LIN {X 0,Y 572.963,Z 565.131,A -85,B 0,C 180,E1 -2344.926,E2 -2344.926} C_VEL
LIN {X 0,Y 573.073,Z 560.098,A -85,B 0,C 180,E1 -2345.984,E2 -2345.984} C_VEL
LIN {X 0,Y 573.083,Z 553.774,A -85,B 0,C 180,E1 -2347.044,E2 -2347.044} C_VEL
LIN {X 0,Y 573.175,Z 545.853,A -85,B 0,C 180,E1 -2348.106,E2 -2348.106} C_VEL
LIN {X 0,Y 573.287,Z 536.003,A -85,B 0,C 180,E1 -2349.17,E2 -2349.17} C_VEL
LIN {X 0,Y 573.412,Z 525.681,A -85,B 0,C 180,E1 -2350.059,E2 -2350.059} C_VEL
LIN {X 0,Y 573.504,Z 514.089,A -85,B 0,C 180,E1 -2350.858,E2 -2350.858} C_VEL
LIN {X 0,Y 573.658,Z 503.195,A -85,B 0,C 180,E1 -2351.449,E2 -2351.449} C_VEL
LIN {X 0,Y 573.732,Z 492.025,A -85,B 0,C 180,E1 -2351.921,E2 -2351.921} C_VEL
LIN {X 0,Y 573.827,Z 479.262,A -85,B 0,C 180,E1 -2352.309,E2 -2352.309} C_VEL
LIN {X 0,Y 573.51,Z 474.932,A -85,B 0,C 180,E1 -2352.417,E2 -2352.417} C_VEL
LIN {X 0,Y 572.962,Z 471.67,A -85,B 0,C 180,E1 -2352.508,E2 -2352.508} C_VEL
LIN {X 0,Y 572.968,Z 468.456,A -85,B 0,C 180,E1 -2354.927,E2 -2354.927} C_VEL
LIN {X 0,Y 572.954,Z 465.205,A -85,B 0,C 180,E1 -2357.402,E2 -2357.402} C_VEL
LIN {X 0,Y 572.988,Z 461.726,A -85,B 0,C 180,E1 -2360.087,E2 -2360.087} C_VEL
LIN {X 0,Y 572.974,Z 461.271,A -85,B 0,C 180,E1 -2360.442,E2 -2360.442} C_VEL
LIN {X 0,Y 572.31,Z 460.562,A -85,B 0,C 180,E1 -2361.024,E2 -2361.024} C_VEL
LIN {X 0,Y 569.449,Z 459.504,A -85,B 0,C 180,E1 -2361.969,E2 -2361.969} C_VEL
LIN {X 0,Y 567.026,Z 458.674,A -85,B 0,C 180,E1 -2362.73,E2 -2362.73} C_VEL
LIN {X 0,Y 565.982,Z 458.008,A -85,B 0,C 180,E1 -2363.318,E2 -2363.318} C_VEL
LIN {X 0,Y 565.895,Z 457.781,A -85,B 0,C 180,E1 -2363.517,E2 -2363.517} C_VEL
LIN {X 0,Y 565.976,Z 454.39,A -85,B 0,C 180,E1 -2366.554,E2 -2366.554} C_VEL
LIN {X 0,Y 565.957,Z 451.602,A -85,B 0,C 180,E1 -2368.967,E2 -2368.967} C_VEL
LIN {X 0,Y 565.973,Z 448.685,A -85,B 0,C 180,E1 -2371.436,E2 -2371.436} C_VEL
LIN {X 0,Y 566.026,Z 445.982,A -85,B 0,C 180,E1 -2373.969,E2 -2373.969} C_VEL
LIN {X 0,Y 566.197,Z 445.959,A -85,B 0,C 180,E1 -2376.571,E2 -2376.571} C_VEL
LIN {X 0,Y 566.218,Z 445.955,A -85,B 0,C 180,E1 -2379.686,E2 -2379.686} C_VEL
LIN {X 0,Y 566.219,Z 445.953,A -85,B 0,C 180,E1 -2382.087,E2 -2382.087} C_VEL
LIN {X 0,Y 566.174,Z 445.959,A -85,B 0,C 180,E1 -2385.036,E2 -2385.036} C_VEL
LIN {X 0,Y 566.194,Z 445.96,A -85,B 0,C 180,E1 -2387.911,E2 -2387.911} C_VEL
LIN {X 0,Y 566.225,Z 445.957,A -85,B 0,C 180,E1 -2390.727,E2 -2390.727} C_VEL
LIN {X 0,Y 566.191,Z 445.96,A -85,B 0,C 180,E1 -2393.788,E2 -2393.788} C_VEL
LIN {X 0,Y 566.219,Z 445.953,A -85,B 0,C 180,E1 -2396.266,E2 -2396.266} C_VEL
LIN {X 0,Y 566.193,Z 445.958,A -85,B 0,C 180,E1 -2398.924,E2 -2398.924} C_VEL
LIN {X 0,Y 566.2,Z 445.96,A -85,B 0,C 180,E1 -2401.856,E2 -2401.856} C_VEL
LIN {X 0,Y 566.22,Z 445.953,A -85,B 0,C 180,E1 -2404.251,E2 -2404.251} C_VEL
LIN {X 0,Y 566.179,Z 445.96,A -85,B 0,C 180,E1 -2406.718,E2 -2406.718} C_VEL
LIN {X 0,Y 566.214,Z 445.958,A -85,B 0,C 180,E1 -2409.663,E2 -2409.663} C_VEL
LIN {X 0,Y 566.206,Z 445.96,A -85,B 0,C 180,E1 -2412.668,E2 -2412.668} C_VEL
LIN {X 0,Y 566.241,Z 445.953,A -85,B 0,C 180,E1 -2415.627,E2 -2415.627} C_VEL
LIN {X 0,Y 566.242,Z 445.953,A -85,B 0,C 180,E1 -2418.675,E2 -2418.675} C_VEL
LIN {X 0,Y 566.211,Z 445.954,A -85,B 0,C 180,E1 -2421.434,E2 -2421.434} C_VEL
LIN {X 0,Y 566.262,Z 445.948,A -85,B 0,C 180,E1 -2424.302,E2 -2424.302} C_VEL
LIN {X 0,Y 566.288,Z 445.946,A -85,B 0,C 180,E1 -2427.866,E2 -2427.866} C_VEL
LIN {X 0,Y 566.306,Z 445.942,A -85,B 0,C 180,E1 -2430.711,E2 -2430.711} C_VEL
LIN {X 0,Y 566.273,Z 445.951,A -85,B 0,C 180,E1 -2432.845,E2 -2432.845} C_VEL
LIN {X 0,Y 566.257,Z 445.95,A -85,B 0,C 180,E1 -2435.698,E2 -2435.698} C_VEL
LIN {X 0,Y 566.234,Z 445.951,A -85,B 0,C 180,E1 -2438.565,E2 -2438.565} C_VEL
LIN {X 0,Y 566.248,Z 445.949,A -85,B 0,C 180,E1 -2441.454,E2 -2441.454} C_VEL
LIN {X 0,Y 566.241,Z 445.95,A -85,B 0,C 180,E1 -2444.506,E2 -2444.506} C_VEL
LIN {X 0,Y 566.205,Z 445.957,A -85,B 0,C 180,E1 -2447.331,E2 -2447.331} C_VEL
LIN {X 0,Y 566.213,Z 445.956,A -85,B 0,C 180,E1 -2450.337,E2 -2450.337} C_VEL
LIN {X 0,Y 566.179,Z 445.963,A -85,B 0,C 180,E1 -2453.282,E2 -2453.282} C_VEL
LIN {X 0,Y 566.218,Z 445.953,A -85,B 0,C 180,E1 -2455.749,E2 -2455.749} C_VEL
LIN {X 0,Y 566.208,Z 445.956,A -85,B 0,C 180,E1 -2458.202,E2 -2458.202} C_VEL
LIN {X 0,Y 566.198,Z 445.961,A -85,B 0,C 180,E1 -2461.076,E2 -2461.076} C_VEL
LIN {X 0,Y 566.217,Z 445.955,A -85,B 0,C 180,E1 -2463.734,E2 -2463.734} C_VEL
LIN {X 0,Y 566.211,Z 445.954,A -85,B 0,C 180,E1 -2466.569,E2 -2466.569} C_VEL
LIN {X 0,Y 566.22,Z 445.953,A -85,B 0,C 180,E1 -2469.686,E2 -2469.686} C_VEL
LIN {X 0,Y 566.205,Z 445.954,A -85,B 0,C 180,E1 -2472.917,E2 -2472.917} C_VEL
LIN {X 0,Y 566.206,Z 445.955,A -85,B 0,C 180,E1 -2476.048,E2 -2476.048} C_VEL
LIN {X 0,Y 566.185,Z 445.957,A -85,B 0,C 180,E1 -2478.861,E2 -2478.861} C_VEL
LIN {X 0,Y 566.188,Z 445.959,A -85,B 0,C 180,E1 -2481.637,E2 -2481.637} C_VEL
LIN {X 0,Y 566.208,Z 445.96,A -85,B 0,C 180,E1 -2484.311,E2 -2484.311} C_VEL
LIN {X 0,Y 566.224,Z 445.952,A -85,B 0,C 180,E1 -2486.898,E2 -2486.898} C_VEL
LIN {X 0,Y 566.187,Z 445.959,A -85,B 0,C 180,E1 -2489.407,E2 -2489.407} C_VEL
LIN {X 0,Y 566.232,Z 445.954,A -85,B 0,C 180,E1 -2491.858,E2 -2491.858} C_VEL
LIN {X 0,Y 566.215,Z 445.954,A -85,B 0,C 180,E1 -2494.251,E2 -2494.251} C_VEL
LIN {X 0,Y 566.175,Z 445.963,A -85,B 0,C 180,E1 -2496.718,E2 -2496.718} C_VEL
LIN {X 0,Y 566.216,Z 445.956,A -85,B 0,C 180,E1 -2499.663,E2 -2499.663} C_VEL
LIN {X 0,Y 566.202,Z 445.956,A -85,B 0,C 180,E1 -2502.668,E2 -2502.668} C_VEL
LIN {X 0,Y 566.237,Z 445.951,A -85,B 0,C 180,E1 -2505.627,E2 -2505.627} C_VEL
LIN {X 0,Y 566.237,Z 445.95,A -85,B 0,C 180,E1 -2508.675,E2 -2508.675} C_VEL
LIN {X 0,Y 566.235,Z 445.952,A -85,B 0,C 180,E1 -2511.434,E2 -2511.434} C_VEL
LIN {X 0,Y 566.259,Z 445.95,A -85,B 0,C 180,E1 -2514.301,E2 -2514.301} C_VEL
LIN {X 0,Y 566.278,Z 445.946,A -85,B 0,C 180,E1 -2517.866,E2 -2517.866} C_VEL
LIN {X 0,Y 566.305,Z 445.943,A -85,B 0,C 180,E1 -2520.711,E2 -2520.711} C_VEL
LIN {X 0,Y 566.275,Z 445.946,A -85,B 0,C 180,E1 -2522.845,E2 -2522.845} C_VEL
LIN {X 0,Y 566.26,Z 445.948,A -85,B 0,C 180,E1 -2525.698,E2 -2525.698} C_VEL
LIN {X 0,Y 566.229,Z 445.952,A -85,B 0,C 180,E1 -2528.566,E2 -2528.566} C_VEL
LIN {X 0,Y 566.244,Z 445.952,A -85,B 0,C 180,E1 -2531.454,E2 -2531.454} C_VEL
LIN {X 0,Y 566.236,Z 445.954,A -85,B 0,C 180,E1 -2534.507,E2 -2534.507} C_VEL
LIN {X 0,Y 566.201,Z 445.96,A -85,B 0,C 180,E1 -2537.332,E2 -2537.332} C_VEL
LIN {X 0,Y 566.216,Z 445.957,A -85,B 0,C 180,E1 -2540.337,E2 -2540.337} C_VEL
LIN {X 0,Y 566.19,Z 445.96,A -85,B 0,C 180,E1 -2543.404,E2 -2543.404} C_VEL
LIN {X 0,Y 566.215,Z 445.954,A -85,B 0,C 180,E1 -2545.749,E2 -2545.749} C_VEL
LIN {X 0,Y 566.203,Z 445.96,A -85,B 0,C 180,E1 -2548.202,E2 -2548.202} C_VEL
LIN {X 0,Y 566.192,Z 445.958,A -85,B 0,C 180,E1 -2551.077,E2 -2551.077} C_VEL
LIN {X 0,Y 566.213,Z 445.954,A -85,B 0,C 180,E1 -2553.734,E2 -2553.734} C_VEL
LIN {X 0,Y 566.216,Z 445.954,A -85,B 0,C 180,E1 -2556.569,E2 -2556.569} C_VEL
LIN {X 0,Y 566.216,Z 445.954,A -85,B 0,C 180,E1 -2559.686,E2 -2559.686} C_VEL
LIN {X 0,Y 566.216,Z 445.956,A -85,B 0,C 180,E1 -2562.087,E2 -2562.087} C_VEL
LIN {X 0,Y 566.17,Z 445.961,A -85,B 0,C 180,E1 -2565.036,E2 -2565.036} C_VEL
LIN {X 0,Y 566.191,Z 445.958,A -85,B 0,C 180,E1 -2567.911,E2 -2567.911} C_VEL
LIN {X 0,Y 566.223,Z 445.954,A -85,B 0,C 180,E1 -2570.727,E2 -2570.727} C_VEL
LIN {X 0,Y 566.236,Z 445.985,A -85,B 0,C 180,E1 -2572.989,E2 -2572.989} C_VEL
LIN {X 0,Y 566.82,Z 449.872,A -85,B 0,C 180,E1 -2574.356,E2 -2574.356} C_VEL
LIN {X 0,Y 566.804,Z 456.508,A -85,B 0,C 180,E1 -2576.554,E2 -2576.554} C_VEL
LIN {X 0,Y 566.648,Z 465.558,A -85,B 0,C 180,E1 -2579.435,E2 -2579.435} C_VEL
LIN {X 0,Y 566.506,Z 476.288,A -85,B 0,C 180,E1 -2582.676,E2 -2582.676} C_VEL
LIN {X 0,Y 566.4,Z 485.661,A -85,B 0,C 180,E1 -2585.438,E2 -2585.438} C_VEL
LIN {X 0,Y 566.323,Z 494.93,A -85,B 0,C 180,E1 -2588.143,E2 -2588.143} C_VEL
LIN {X 0,Y 566.185,Z 505.521,A -85,B 0,C 180,E1 -2591.172,E2 -2591.172} C_VEL
LIN {X 0,Y 566.116,Z 516.112,A -85,B 0,C 180,E1 -2594.15,E2 -2594.15} C_VEL
LIN {X 0,Y 566.058,Z 525.379,A -85,B 0,C 180,E1 -2596.721,E2 -2596.721} C_VEL
LIN {X 0,Y 566.033,Z 527.531,A -85,B 0,C 180,E1 -2597.314,E2 -2597.314} C_VEL
LIN {X 0,Y 566.941,Z 534.376,A -85,B 0,C 180,E1 -2597.471,E2 -2597.471} C_VEL
LIN {X 0,Y 566.856,Z 546.503,A -85,B 0,C 180,E1 -2597.787,E2 -2597.787} C_VEL
LIN {X 0,Y 566.719,Z 558.32,A -85,B 0,C 180,E1 -2598.229,E2 -2598.229} C_VEL
LIN {X 0,Y 566.571,Z 570.729,A -85,B 0,C 180,E1 -2598.854,E2 -2598.854} C_VEL
LIN {X 0,Y 566.418,Z 581.483,A -85,B 0,C 180,E1 -2599.545,E2 -2599.545} C_VEL
LIN {X 0,Y 566.301,Z 591.648,A -85,B 0,C 180,E1 -2600.355,E2 -2600.355} C_VEL
LIN {X 0,Y 566.166,Z 600.788,A -85,B 0,C 180,E1 -2601.254,E2 -2601.254} C_VEL
LIN {X 0,Y 566.08,Z 609.691,A -85,B 0,C 180,E1 -2602.33,E2 -2602.33} C_VEL
LIN {X 0,Y 565.967,Z 616.956,A -85,B 0,C 180,E1 -2603.422,E2 -2603.422} C_VEL
LIN {X 0,Y 566.004,Z 621.681,A -85,B 0,C 180,E1 -2604.299,E2 -2604.299} C_VEL
LIN {X 0,Y 565.933,Z 626.373,A -85,B 0,C 180,E1 -2605.37,E2 -2605.37} C_VEL
LIN {X 0,Y 565.927,Z 629.958,A -85,B 0,C 180,E1 -2606.44,E2 -2606.44} C_VEL
LIN {X 0,Y 565.878,Z 631.809,A -85,B 0,C 180,E1 -2607.153,E2 -2607.153} C_VEL
LIN {X 0,Y 565.846,Z 634.186,A -85,B 0,C 180,E1 -2608.577,E2 -2608.577} C_VEL
LIN {X 0,Y 565.839,Z 635,A -85,B 0,C 180,E1 -2610,E2 -2610} C_VEL
LIN {X 0,Y 565.846,Z 634.186,A -85,B 0,C 180,E1 -2611.424,E2 -2611.424} C_VEL
LIN {X 0,Y 565.878,Z 631.809,A -85,B 0,C 180,E1 -2612.848,E2 -2612.848} C_VEL
LIN {X 0,Y 565.926,Z 628.895,A -85,B 0,C 180,E1 -2613.917,E2 -2613.917} C_VEL
LIN {X 0,Y 565.878,Z 624.948,A -85,B 0,C 180,E1 -2614.988,E2 -2614.988} C_VEL
LIN {X 0,Y 566.002,Z 619.866,A -85,B 0,C 180,E1 -2616.059,E2 -2616.059} C_VEL
LIN {X 0,Y 566.04,Z 613.467,A -85,B 0,C 180,E1 -2617.132,E2 -2617.132} C_VEL
LIN {X 0,Y 566.134,Z 605.477,A -85,B 0,C 180,E1 -2618.208,E2 -2618.208} C_VEL
LIN {X 0,Y 566.229,Z 597.334,A -85,B 0,C 180,E1 -2619.106,E2 -2619.106} C_VEL
LIN {X 0,Y 566.343,Z 587.399,A -85,B 0,C 180,E1 -2620.005,E2 -2620.005} C_VEL
LIN {X 0,Y 566.535,Z 576.295,A -85,B 0,C 180,E1 -2620.807,E2 -2620.807} C_VEL
LIN {X 0,Y 566.613,Z 565.174,A -85,B 0,C 180,E1 -2621.447,E2 -2621.447} C_VEL
LIN {X 0,Y 566.75,Z 552.98,A -85,B 0,C 180,E1 -2621.988,E2 -2621.988} C_VEL
LIN {X 0,Y 566.881,Z 540.169,A -85,B 0,C 180,E1 -2622.394,E2 -2622.394} C_VEL
LIN {X 0,Y 566.748,Z 532.075,A -85,B 0,C 180,E1 -2622.579,E2 -2622.579} C_VEL
LIN {X 0,Y 566.033,Z 527.529,A -85,B 0,C 180,E1 -2622.686,E2 -2622.686} C_VEL
LIN {X 0,Y 566.091,Z 517.435,A -85,B 0,C 180,E1 -2625.481,E2 -2625.481} C_VEL
LIN {X 0,Y 566.167,Z 506.844,A -85,B 0,C 180,E1 -2628.454,E2 -2628.454} C_VEL
LIN {X 0,Y 566.245,Z 497.576,A -85,B 0,C 180,E1 -2631.096,E2 -2631.096} C_VEL
LIN {X 0,Y 566.362,Z 488.309,A -85,B 0,C 180,E1 -2633.784,E2 -2633.784} C_VEL
LIN {X 0,Y 566.426,Z 480.094,A -85,B 0,C 180,E1 -2636.134,E2 -2636.134} C_VEL
LIN {X 0,Y 566.448,Z 471.713,A -85,B 0,C 180,E1 -2638.557,E2 -2638.557} C_VEL
LIN {X 0,Y 566.56,Z 463.235,A -85,B 0,C 180,E1 -2641.138,E2 -2641.138} C_VEL
LIN {X 0,Y 566.718,Z 455.161,A -85,B 0,C 180,E1 -2643.81,E2 -2643.81} C_VEL
LIN {X 0,Y 566.858,Z 450.195,A -85,B 0,C 180,E1 -2645.642,E2 -2645.642} C_VEL
LIN {X 0,Y 566.22,Z 445.959,A -85,B 0,C 180,E1 -2647.571,E2 -2647.571} C_VEL
LIN {X 0,Y 566.231,Z 445.957,A -85,B 0,C 180,E1 -2650.197,E2 -2650.197} C_VEL
LIN {X 0,Y 566.204,Z 445.958,A -85,B 0,C 180,E1 -2653.054,E2 -2653.054} C_VEL
LIN {X 0,Y 566.206,Z 445.96,A -85,B 0,C 180,E1 -2656.048,E2 -2656.048} C_VEL
LIN {X 0,Y 566.215,Z 445.958,A -85,B 0,C 180,E1 -2658.864,E2 -2658.864} C_VEL
LIN {X 0,Y 566.194,Z 445.959,A -85,B 0,C 180,E1 -2661.637,E2 -2661.637} C_VEL
LIN {X 0,Y 566.137,Z 445.967,A -85,B 0,C 180,E1 -2664.306,E2 -2664.306} C_VEL
LIN {X 0,Y 566.127,Z 446.063,A -85,B 0,C 180,E1 -2665.176,E2 -2665.176} C_VEL
LIN {X 0,Y 566.103,Z 448.7,A -85,B 0,C 180,E1 -2667.735,E2 -2667.735} C_VEL
LIN {X 0,Y 566.046,Z 451.422,A -85,B 0,C 180,E1 -2670.357,E2 -2670.357} C_VEL
LIN {X 0,Y 566.001,Z 454.553,A -85,B 0,C 180,E1 -2673.448,E2 -2673.448} C_VEL
LIN {X 0,Y 565.923,Z 456.995,A -85,B 0,C 180,E1 -2675.807,E2 -2675.807} C_VEL
LIN {X 0,Y 565.906,Z 460.651,A -85,B 0,C 180,E1 -2678.891,E2 -2678.891} C_VEL
LIN {X 0,Y 565.866,Z 464.495,A -85,B 0,C 180,E1 -2681.911,E2 -2681.911} C_VEL
LIN {X 0,Y 565.89,Z 468.338,A -85,B 0,C 180,E1 -2684.882,E2 -2684.882} C_VEL
LIN {X 0,Y 565.873,Z 471.671,A -85,B 0,C 180,E1 -2687.424,E2 -2687.424} C_VEL
LIN {X 0,Y 566.904,Z 479.284,A -85,B 0,C 180,E1 -2687.629,E2 -2687.629} C_VEL
LIN {X 0,Y 566.781,Z 491.783,A -85,B 0,C 180,E1 -2688.013,E2 -2688.013} C_VEL
LIN {X 0,Y 566.661,Z 504.301,A -85,B 0,C 180,E1 -2688.554,E2 -2688.554} C_VEL
LIN {X 0,Y 566.543,Z 515.586,A -85,B 0,C 180,E1 -2689.193,E2 -2689.193} C_VEL
LIN {X 0,Y 566.341,Z 526.843,A -85,B 0,C 180,E1 -2689.995,E2 -2689.995} C_VEL
LIN {X 0,Y 566.238,Z 536.892,A -85,B 0,C 180,E1 -2690.895,E2 -2690.895} C_VEL
LIN {X 0,Y 566.113,Z 546.592,A -85,B 0,C 180,E1 -2691.972,E2 -2691.972} C_VEL
LIN {X 0,Y 566.05,Z 553.16,A -85,B 0,C 180,E1 -2692.868,E2 -2692.868} C_VEL
LIN {X 0,Y 566.003,Z 559.628,A -85,B 0,C 180,E1 -2693.942,E2 -2693.942} C_VEL
LIN {X 0,Y 565.878,Z 564.765,A -85,B 0,C 180,E1 -2695.013,E2 -2695.013} C_VEL
LIN {X 0,Y 565.926,Z 568.754,A -85,B 0,C 180,E1 -2696.084,E2 -2696.084} C_VEL
LIN {X 0,Y 565.878,Z 571.702,A -85,B 0,C 180,E1 -2697.153,E2 -2697.153} C_VEL
LIN {X 0,Y 565.839,Z 573.129,A -85,B 0,C 180,E1 -2697.865,E2 -2697.865} C_VEL
LIN {X 0,Y 565.841,Z 574.756,A -85,B 0,C 180,E1 -2699.289,E2 -2699.289} C_VEL
LIN {X 0,Y 565.839,Z 574.996,A -85,B 0,C 180,E1 -2700,E2 -2700} C_VEL
LIN {X 0,Y 565.841,Z 574.814,A -85,B 0,C 180,E1 -2700.712,E2 -2700.712} C_VEL
LIN {X 0,Y 565.838,Z 573.269,A -85,B 0,C 180,E1 -2702.136,E2 -2702.136} C_VEL
LIN {X 0,Y 565.878,Z 571.907,A -85,B 0,C 180,E1 -2702.848,E2 -2702.848} C_VEL
LIN {X 0,Y 565.926,Z 569.029,A -85,B 0,C 180,E1 -2703.917,E2 -2703.917} C_VEL
LIN {X 0,Y 565.878,Z 565.128,A -85,B 0,C 180,E1 -2704.988,E2 -2704.988} C_VEL
LIN {X 0,Y 565.988,Z 560.095,A -85,B 0,C 180,E1 -2706.059,E2 -2706.059} C_VEL
LIN {X 0,Y 566.031,Z 553.771,A -85,B 0,C 180,E1 -2707.133,E2 -2707.133} C_VEL
LIN {X 0,Y 566.128,Z 545.848,A -85,B 0,C 180,E1 -2708.208,E2 -2708.208} C_VEL
LIN {X 0,Y 566.249,Z 535.997,A -85,B 0,C 180,E1 -2709.285,E2 -2709.285} C_VEL
LIN {X 0,Y 566.413,Z 525.675,A -85,B 0,C 180,E1 -2710.184,E2 -2710.184} C_VEL
LIN {X 0,Y 566.519,Z 514.394,A -85,B 0,C 180,E1 -2710.973,E2 -2710.973} C_VEL
LIN {X 0,Y 566.688,Z 503.183,A -85,B 0,C 180,E1 -2711.592,E2 -2711.592} C_VEL
LIN {X 0,Y 566.786,Z 492.009,A -85,B 0,C 180,E1 -2712.069,E2 -2712.069} C_VEL
LIN {X 0,Y 566.896,Z 479.239,A -85,B 0,C 180,E1 -2712.462,E2 -2712.462} C_VEL
LIN {X 0,Y 565.878,Z 471.669,A -85,B 0,C 180,E1 -2712.667,E2 -2712.667} C_VEL
LIN {X 0,Y 565.891,Z 468.455,A -85,B 0,C 180,E1 -2715.118,E2 -2715.118} C_VEL
LIN {X 0,Y 565.868,Z 464.61,A -85,B 0,C 180,E1 -2718.089,E2 -2718.089} C_VEL
LIN {X 0,Y 565.906,Z 460.764,A -85,B 0,C 180,E1 -2721.11,E2 -2721.11} C_VEL
LIN {X 0,Y 565.895,Z 457.781,A -85,B 0,C 180,E1 -2723.517,E2 -2723.517} C_VEL
LIN {X 0,Y 565.218,Z 457.167,A -85,B 0,C 180,E1 -2724.107,E2 -2724.107} C_VEL
LIN {X 0,Y 562.35,Z 456.326,A -85,B 0,C 180,E1 -2725.068,E2 -2725.068} C_VEL
LIN {X 0,Y 559.956,Z 455.672,A -85,B 0,C 180,E1 -2725.842,E2 -2725.842} C_VEL
LIN {X 0,Y 558.962,Z 455.108,A -85,B 0,C 180,E1 -2726.438,E2 -2726.438} C_VEL
LIN {X 0,Y 558.898,Z 454.896,A -85,B 0,C 180,E1 -2726.639,E2 -2726.639} C_VEL
LIN {X 0,Y 558.904,Z 451.659,A -85,B 0,C 180,E1 -2729.368,E2 -2729.368} C_VEL
LIN {X 0,Y 558.901,Z 448.772,A -85,B 0,C 180,E1 -2731.88,E2 -2731.88} C_VEL
LIN {X 0,Y 558.928,Z 446.866,A -85,B 0,C 180,E1 -2733.591,E2 -2733.591} C_VEL
LIN {X 0,Y 559.141,Z 446.837,A -85,B 0,C 180,E1 -2736.444,E2 -2736.444} C_VEL
LIN {X 0,Y 559.177,Z 446.83,A -85,B 0,C 180,E1 -2738.934,E2 -2738.934} C_VEL
LIN {X 0,Y 559.182,Z 446.83,A -85,B 0,C 180,E1 -2742.137,E2 -2742.137} C_VEL
LIN {X 0,Y 559.14,Z 446.834,A -85,B 0,C 180,E1 -2745.261,E2 -2745.261} C_VEL
LIN {X 0,Y 559.168,Z 446.832,A -85,B 0,C 180,E1 -2748.23,E2 -2748.23} C_VEL
LIN {X 0,Y 559.182,Z 446.831,A -85,B 0,C 180,E1 -2751.192,E2 -2751.192} C_VEL
LIN {X 0,Y 559.146,Z 446.837,A -85,B 0,C 180,E1 -2753.789,E2 -2753.789} C_VEL
LIN {X 0,Y 559.169,Z 446.831,A -85,B 0,C 180,E1 -2756.425,E2 -2756.425} C_VEL
LIN {X 0,Y 559.157,Z 446.834,A -85,B 0,C 180,E1 -2758.981,E2 -2758.981} C_VEL
LIN {X 0,Y 559.151,Z 446.837,A -85,B 0,C 180,E1 -2761.623,E2 -2761.623} C_VEL
LIN {X 0,Y 559.187,Z 446.829,A -85,B 0,C 180,E1 -2763.903,E2 -2763.903} C_VEL
LIN {X 0,Y 559.149,Z 446.837,A -85,B 0,C 180,E1 -2766.571,E2 -2766.571} C_VEL
LIN {X 0,Y 559.183,Z 446.833,A -85,B 0,C 180,E1 -2769.395,E2 -2769.395} C_VEL
LIN {X 0,Y 559.148,Z 446.834,A -85,B 0,C 180,E1 -2771.686,E2 -2771.686} C_VEL
LIN {X 0,Y 559.167,Z 446.834,A -85,B 0,C 180,E1 -2773.948,E2 -2773.948} C_VEL
LIN {X 0,Y 559.178,Z 446.831,A -85,B 0,C 180,E1 -2776.184,E2 -2776.184} C_VEL
LIN {X 0,Y 559.201,Z 446.83,A -85,B 0,C 180,E1 -2779.133,E2 -2779.133} C_VEL
LIN {X 0,Y 559.198,Z 446.833,A -85,B 0,C 180,E1 -2782.053,E2 -2782.053} C_VEL
LIN {X 0,Y 559.256,Z 446.824,A -85,B 0,C 180,E1 -2784.953,E2 -2784.953} C_VEL
LIN {X 0,Y 559.259,Z 446.821,A -85,B 0,C 180,E1 -2787.839,E2 -2787.839} C_VEL
LIN {X 0,Y 559.277,Z 446.818,A -85,B 0,C 180,E1 -2790.72,E2 -2790.72} C_VEL
LIN {X 0,Y 559.24,Z 446.827,A -85,B 0,C 180,E1 -2792.881,E2 -2792.881} C_VEL
LIN {X 0,Y 559.225,Z 446.826,A -85,B 0,C 180,E1 -2795.77,E2 -2795.77} C_VEL
LIN {X 0,Y 559.193,Z 446.829,A -85,B 0,C 180,E1 -2798.674,E2 -2798.674} C_VEL
LIN {X 0,Y 559.212,Z 446.826,A -85,B 0,C 180,E1 -2801.6,E2 -2801.6} C_VEL
LIN {X 0,Y 559.207,Z 446.826,A -85,B 0,C 180,E1 -2804.595,E2 -2804.595} C_VEL
LIN {X 0,Y 559.164,Z 446.832,A -85,B 0,C 180,E1 -2807.557,E2 -2807.557} C_VEL
LIN {X 0,Y 559.171,Z 446.834,A -85,B 0,C 180,E1 -2809.837,E2 -2809.837} C_VEL
LIN {X 0,Y 559.146,Z 446.835,A -85,B 0,C 180,E1 -2812.153,E2 -2812.153} C_VEL
LIN {X 0,Y 559.181,Z 446.83,A -85,B 0,C 180,E1 -2815.298,E2 -2815.298} C_VEL
LIN {X 0,Y 559.173,Z 446.831,A -85,B 0,C 180,E1 -2818.381,E2 -2818.381} C_VEL
LIN {X 0,Y 559.153,Z 446.836,A -85,B 0,C 180,E1 -2821.273,E2 -2821.273} C_VEL
LIN {X 0,Y 559.172,Z 446.835,A -85,B 0,C 180,E1 -2823.949,E2 -2823.949} C_VEL
LIN {X 0,Y 559.147,Z 446.838,A -85,B 0,C 180,E1 -2827.108,E2 -2827.108} C_VEL
LIN {X 0,Y 559.165,Z 446.833,A -85,B 0,C 180,E1 -2829.941,E2 -2829.941} C_VEL
LIN {X 0,Y 559.16,Z 446.831,A -85,B 0,C 180,E1 -2832.743,E2 -2832.743} C_VEL
LIN {X 0,Y 559.159,Z 446.833,A -85,B 0,C 180,E1 -2835.76,E2 -2835.76} C_VEL
LIN {X 0,Y 559.192,Z 446.833,A -85,B 0,C 180,E1 -2838.232,E2 -2838.232} C_VEL
LIN {X 0,Y 559.177,Z 446.834,A -85,B 0,C 180,E1 -2841.191,E2 -2841.191} C_VEL
LIN {X 0,Y 559.173,Z 446.831,A -85,B 0,C 180,E1 -2843.791,E2 -2843.791} C_VEL
LIN {X 0,Y 559.165,Z 446.832,A -85,B 0,C 180,E1 -2846.425,E2 -2846.425} C_VEL
LIN {X 0,Y 559.162,Z 446.836,A -85,B 0,C 180,E1 -2848.981,E2 -2848.981} C_VEL
LIN {X 0,Y 559.171,Z 446.831,A -85,B 0,C 180,E1 -2851.618,E2 -2851.618} C_VEL
LIN {X 0,Y 559.183,Z 446.833,A -85,B 0,C 180,E1 -2853.903,E2 -2853.903} C_VEL
LIN {X 0,Y 559.145,Z 446.837,A -85,B 0,C 180,E1 -2856.571,E2 -2856.571} C_VEL
LIN {X 0,Y 559.182,Z 446.83,A -85,B 0,C 180,E1 -2859.395,E2 -2859.395} C_VEL
LIN {X 0,Y 559.146,Z 446.838,A -85,B 0,C 180,E1 -2861.685,E2 -2861.685} C_VEL
LIN {X 0,Y 559.169,Z 446.831,A -85,B 0,C 180,E1 -2863.948,E2 -2863.948} C_VEL
LIN {X 0,Y 559.175,Z 446.836,A -85,B 0,C 180,E1 -2866.184,E2 -2866.184} C_VEL
LIN {X 0,Y 559.196,Z 446.83,A -85,B 0,C 180,E1 -2869.133,E2 -2869.133} C_VEL
LIN {X 0,Y 559.207,Z 446.828,A -85,B 0,C 180,E1 -2872.053,E2 -2872.053} C_VEL
LIN {X 0,Y 559.256,Z 446.82,A -85,B 0,C 180,E1 -2874.953,E2 -2874.953} C_VEL
LIN {X 0,Y 559.25,Z 446.821,A -85,B 0,C 180,E1 -2877.839,E2 -2877.839} C_VEL
LIN {X 0,Y 559.275,Z 446.819,A -85,B 0,C 180,E1 -2880.72,E2 -2880.72} C_VEL
LIN {X 0,Y 559.241,Z 446.822,A -85,B 0,C 180,E1 -2882.881,E2 -2882.881} C_VEL
LIN {X 0,Y 559.229,Z 446.824,A -85,B 0,C 180,E1 -2885.77,E2 -2885.77} C_VEL
LIN {X 0,Y 559.188,Z 446.829,A -85,B 0,C 180,E1 -2888.674,E2 -2888.674} C_VEL
LIN {X 0,Y 559.207,Z 446.828,A -85,B 0,C 180,E1 -2891.6,E2 -2891.6} C_VEL
LIN {X 0,Y 559.201,Z 446.829,A -85,B 0,C 180,E1 -2894.595,E2 -2894.595} C_VEL
LIN {X 0,Y 559.161,Z 446.836,A -85,B 0,C 180,E1 -2897.557,E2 -2897.557} C_VEL
LIN {X 0,Y 559.174,Z 446.831,A -85,B 0,C 180,E1 -2899.837,E2 -2899.837} C_VEL
LIN {X 0,Y 559.144,Z 446.839,A -85,B 0,C 180,E1 -2902.153,E2 -2902.153} C_VEL
LIN {X 0,Y 559.177,Z 446.835,A -85,B 0,C 180,E1 -2905.298,E2 -2905.298} C_VEL
LIN {X 0,Y 559.182,Z 446.83,A -85,B 0,C 180,E1 -2907.712,E2 -2907.712} C_VEL
LIN {X 0,Y 559.155,Z 446.835,A -85,B 0,C 180,E1 -2910.183,E2 -2910.183} C_VEL
LIN {X 0,Y 559.158,Z 446.834,A -85,B 0,C 180,E1 -2912.715,E2 -2912.715} C_VEL
LIN {X 0,Y 559.15,Z 446.834,A -85,B 0,C 180,E1 -2915.323,E2 -2915.323} C_VEL
LIN {X 0,Y 559.134,Z 446.837,A -85,B 0,C 180,E1 -2918.018,E2 -2918.018} C_VEL
LIN {X 0,Y 559.163,Z 446.837,A -85,B 0,C 180,E1 -2920.812,E2 -2920.812} C_VEL
LIN {X 0,Y 559.164,Z 446.836,A -85,B 0,C 180,E1 -2923.732,E2 -2923.732} C_VEL
LIN {X 0,Y 559.146,Z 446.839,A -85,B 0,C 180,E1 -2926.804,E2 -2926.804} C_VEL
LIN {X 0,Y 559.175,Z 446.832,A -85,B 0,C 180,E1 -2929.189,E2 -2929.189} C_VEL
LIN {X 0,Y 559.136,Z 446.84,A -85,B 0,C 180,E1 -2931.983,E2 -2931.983} C_VEL
LIN {X 0,Y 559.215,Z 447.004,A -85,B 0,C 180,E1 -2932.8,E2 -2932.8} C_VEL
LIN {X 0,Y 559.892,Z 452.465,A -85,B 0,C 180,E1 -2934.731,E2 -2934.731} C_VEL
LIN {X 0,Y 559.772,Z 460.095,A -85,B 0,C 180,E1 -2937.267,E2 -2937.267} C_VEL
LIN {X 0,Y 559.625,Z 468.857,A -85,B 0,C 180,E1 -2940.058,E2 -2940.058} C_VEL
LIN {X 0,Y 559.467,Z 478.897,A -85,B 0,C 180,E1 -2943.113,E2 -2943.113} C_VEL
LIN {X 0,Y 559.379,Z 488.262,A -85,B 0,C 180,E1 -2945.9,E2 -2945.9} C_VEL
LIN {X 0,Y 559.233,Z 497.577,A -85,B 0,C 180,E1 -2948.626,E2 -2948.626} C_VEL
LIN {X 0,Y 559.134,Z 506.845,A -85,B 0,C 180,E1 -2951.306,E2 -2951.306} C_VEL
LIN {X 0,Y 559.055,Z 517.436,A -85,B 0,C 180,E1 -2954.319,E2 -2954.319} C_VEL
LIN {X 0,Y 558.955,Z 527.531,A -85,B 0,C 180,E1 -2957.151,E2 -2957.151} C_VEL
LIN {X 0,Y 560.015,Z 535.515,A -85,B 0,C 180,E1 -2957.336,E2 -2957.336} C_VEL
LIN {X 0,Y 559.897,Z 547.879,A -85,B 0,C 180,E1 -2957.679,E2 -2957.679} C_VEL
LIN {X 0,Y 559.759,Z 560.285,A -85,B 0,C 180,E1 -2958.172,E2 -2958.172} C_VEL
LIN {X 0,Y 559.608,Z 572.583,A -85,B 0,C 180,E1 -2958.822,E2 -2958.822} C_VEL
LIN {X 0,Y 559.425,Z 583.926,A -85,B 0,C 180,E1 -2959.596,E2 -2959.596} C_VEL
LIN {X 0,Y 559.243,Z 593.602,A -85,B 0,C 180,E1 -2960.415,E2 -2960.415} C_VEL
LIN {X 0,Y 559.127,Z 602.414,A -85,B 0,C 180,E1 -2961.325,E2 -2961.325} C_VEL
LIN {X 0,Y 558.996,Z 611.003,A -85,B 0,C 180,E1 -2962.414,E2 -2962.414} C_VEL
LIN {X 0,Y 558.884,Z 618.688,A -85,B 0,C 180,E1 -2963.649,E2 -2963.649} C_VEL
LIN {X 0,Y 558.869,Z 623.366,A -85,B 0,C 180,E1 -2964.588,E2 -2964.588} C_VEL
LIN {X 0,Y 558.868,Z 627.678,A -85,B 0,C 180,E1 -2965.673,E2 -2965.673} C_VEL
LIN {X 0,Y 558.836,Z 629.958,A -85,B 0,C 180,E1 -2966.395,E2 -2966.395} C_VEL
LIN {X 0,Y 558.799,Z 631.808,A -85,B 0,C 180,E1 -2967.117,E2 -2967.117} C_VEL
LIN {X 0,Y 558.745,Z 634.185,A -85,B 0,C 180,E1 -2968.559,E2 -2968.559} C_VEL
LIN {X 0,Y 558.74,Z 635,A -85,B 0,C 180,E1 -2970,E2 -2970} C_VEL
LIN {X 0,Y 558.745,Z 634.186,A -85,B 0,C 180,E1 -2971.442,E2 -2971.442} C_VEL
LIN {X 0,Y 558.799,Z 631.81,A -85,B 0,C 180,E1 -2972.884,E2 -2972.884} C_VEL
LIN {X 0,Y 558.843,Z 628.895,A -85,B 0,C 180,E1 -2973.966,E2 -2973.966} C_VEL
LIN {X 0,Y 558.799,Z 624.948,A -85,B 0,C 180,E1 -2975.051,E2 -2975.051} C_VEL
LIN {X 0,Y 558.921,Z 619.866,A -85,B 0,C 180,E1 -2976.136,E2 -2976.136} C_VEL
LIN {X 0,Y 558.977,Z 613.467,A -85,B 0,C 180,E1 -2977.223,E2 -2977.223} C_VEL
LIN {X 0,Y 559.099,Z 605.477,A -85,B 0,C 180,E1 -2978.312,E2 -2978.312} C_VEL
LIN {X 0,Y 559.195,Z 597.333,A -85,B 0,C 180,E1 -2979.221,E2 -2979.221} C_VEL
LIN {X 0,Y 559.351,Z 587.398,A -85,B 0,C 180,E1 -2980.131,E2 -2980.131} C_VEL
LIN {X 0,Y 559.538,Z 576.398,A -85,B 0,C 180,E1 -2980.937,E2 -2980.937} C_VEL
LIN {X 0,Y 559.672,Z 564.458,A -85,B 0,C 180,E1 -2981.628,E2 -2981.628} C_VEL
LIN {X 0,Y 559.824,Z 551.762,A -85,B 0,C 180,E1 -2982.185,E2 -2982.185} C_VEL
LIN {X 0,Y 559.974,Z 538.339,A -85,B 0,C 180,E1 -2982.596,E2 -2982.596} C_VEL
LIN {X 0,Y 559.749,Z 532.507,A -85,B 0,C 180,E1 -2982.73,E2 -2982.73} C_VEL
LIN {X 0,Y 558.955,Z 527.529,A -85,B 0,C 180,E1 -2982.85,E2 -2982.85} C_VEL
LIN {X 0,Y 559.055,Z 517.435,A -85,B 0,C 180,E1 -2985.681,E2 -2985.681} C_VEL
LIN {X 0,Y 559.134,Z 506.844,A -85,B 0,C 180,E1 -2988.695,E2 -2988.695} C_VEL
LIN {X 0,Y 559.227,Z 496.916,A -85,B 0,C 180,E1 -2991.567,E2 -2991.567} C_VEL
LIN {X 0,Y 559.345,Z 488.126,A -85,B 0,C 180,E1 -2994.102,E2 -2994.102} C_VEL
LIN {X 0,Y 559.42,Z 478.359,A -85,B 0,C 180,E1 -2996.89,E2 -2996.89} C_VEL
LIN {X 0,Y 559.529,Z 468.262,A -85,B 0,C 180,E1 -2999.925,E2 -2999.925} C_VEL
LIN {X 0,Y 559.677,Z 459.655,A -85,B 0,C 180,E1 -3002.718,E2 -3002.718} C_VEL
LIN {X 0,Y 559.896,Z 452.496,A -85,B 0,C 180,E1 -3005.323,E2 -3005.323} C_VEL
LIN {X 0,Y 559.691,Z 449.63,A -85,B 0,C 180,E1 -3006.52,E2 -3006.52} C_VEL
LIN {X 0,Y 559.169,Z 446.837,A -85,B 0,C 180,E1 -3007.907,E2 -3007.907} C_VEL
LIN {X 0,Y 559.177,Z 446.834,A -85,B 0,C 180,E1 -3010.811,E2 -3010.811} C_VEL
LIN {X 0,Y 559.144,Z 446.84,A -85,B 0,C 180,E1 -3013.734,E2 -3013.734} C_VEL
LIN {X 0,Y 559.172,Z 446.834,A -85,B 0,C 180,E1 -3016.801,E2 -3016.801} C_VEL
LIN {X 0,Y 559.18,Z 446.833,A -85,B 0,C 180,E1 -3019.19,E2 -3019.19} C_VEL
LIN {X 0,Y 559.139,Z 446.839,A -85,B 0,C 180,E1 -3021.983,E2 -3021.983} C_VEL
LIN {X 0,Y 559.075,Z 446.849,A -85,B 0,C 180,E1 -3024.672,E2 -3024.672} C_VEL
LIN {X 0,Y 559.059,Z 448.217,A -85,B 0,C 180,E1 -3026.418,E2 -3026.418} C_VEL
LIN {X 0,Y 559.03,Z 450.796,A -85,B 0,C 180,E1 -3028.973,E2 -3028.973} C_VEL
LIN {X 0,Y 558.95,Z 453.54,A -85,B 0,C 180,E1 -3031.661,E2 -3031.661} C_VEL
LIN {X 0,Y 558.896,Z 456.578,A -85,B 0,C 180,E1 -3034.688,E2 -3034.688} C_VEL
LIN {X 0,Y 558.816,Z 459.044,A -85,B 0,C 180,E1 -3037.053,E2 -3037.053} C_VEL
LIN {X 0,Y 558.789,Z 461.613,A -85,B 0,C 180,E1 -3039.38,E2 -3039.38} C_VEL
LIN {X 0,Y 558.764,Z 464.495,A -85,B 0,C 180,E1 -3041.673,E2 -3041.673} C_VEL
LIN {X 0,Y 558.773,Z 467.378,A -85,B 0,C 180,E1 -3043.936,E2 -3043.936} C_VEL
LIN {X 0,Y 558.782,Z 470.261,A -85,B 0,C 180,E1 -3046.174,E2 -3046.174} C_VEL
LIN {X 0,Y 558.784,Z 471.672,A -85,B 0,C 180,E1 -3047.262,E2 -3047.262} C_VEL
LIN {X 0,Y 559.972,Z 480.22,A -85,B 0,C 180,E1 -3047.497,E2 -3047.497} C_VEL
LIN {X 0,Y 559.835,Z 492.301,A -85,B 0,C 180,E1 -3047.88,E2 -3047.88} C_VEL
LIN {X 0,Y 559.688,Z 504.311,A -85,B 0,C 180,E1 -3048.41,E2 -3048.41} C_VEL
LIN {X 0,Y 559.566,Z 515.668,A -85,B 0,C 180,E1 -3049.061,E2 -3049.061} C_VEL
LIN {X 0,Y 559.356,Z 526.851,A -85,B 0,C 180,E1 -3049.869,E2 -3049.869} C_VEL
LIN {X 0,Y 559.21,Z 536.897,A -85,B 0,C 180,E1 -3050.779,E2 -3050.779} C_VEL
LIN {X 0,Y 559.05,Z 546.596,A -85,B 0,C 180,E1 -3051.87,E2 -3051.87} C_VEL
LIN {X 0,Y 558.971,Z 554.456,A -85,B 0,C 180,E1 -3052.977,E2 -3052.977} C_VEL
LIN {X 0,Y 558.936,Z 561.455,A -85,B 0,C 180,E1 -3054.227,E2 -3054.227} C_VEL
LIN {X 0,Y 558.826,Z 566.195,A -85,B 0,C 180,E1 -3055.311,E2 -3055.311} C_VEL
LIN {X 0,Y 558.837,Z 569.828,A -85,B 0,C 180,E1 -3056.395,E2 -3056.395} C_VEL
LIN {X 0,Y 558.799,Z 571.704,A -85,B 0,C 180,E1 -3057.117,E2 -3057.117} C_VEL
LIN {X 0,Y 558.745,Z 573.129,A -85,B 0,C 180,E1 -3057.838,E2 -3057.838} C_VEL
LIN {X 0,Y 558.742,Z 574.757,A -85,B 0,C 180,E1 -3059.279,E2 -3059.279} C_VEL
LIN {X 0,Y 558.74,Z 574.996,A -85,B 0,C 180,E1 -3060,E2 -3060} C_VEL
LIN {X 0,Y 558.741,Z 574.814,A -85,B 0,C 180,E1 -3060.721,E2 -3060.721} C_VEL
LIN {X 0,Y 558.745,Z 573.267,A -85,B 0,C 180,E1 -3062.163,E2 -3062.163} C_VEL
LIN {X 0,Y 558.8,Z 571.905,A -85,B 0,C 180,E1 -3062.884,E2 -3062.884} C_VEL
LIN {X 0,Y 558.844,Z 569.028,A -85,B 0,C 180,E1 -3063.966,E2 -3063.966} C_VEL
LIN {X 0,Y 558.798,Z 565.126,A -85,B 0,C 180,E1 -3065.051,E2 -3065.051} C_VEL
LIN {X 0,Y 558.908,Z 560.093,A -85,B 0,C 180,E1 -3066.136,E2 -3066.136} C_VEL
LIN {X 0,Y 558.973,Z 553.767,A -85,B 0,C 180,E1 -3067.223,E2 -3067.223} C_VEL
LIN {X 0,Y 559.091,Z 545.843,A -85,B 0,C 180,E1 -3068.312,E2 -3068.312} C_VEL
LIN {X 0,Y 559.224,Z 535.99,A -85,B 0,C 180,E1 -3069.403,E2 -3069.403} C_VEL
LIN {X 0,Y 559.399,Z 525.669,A -85,B 0,C 180,E1 -3070.313,E2 -3070.313} C_VEL
LIN {X 0,Y 559.533,Z 514.701,A -85,B 0,C 180,E1 -3071.091,E2 -3071.091} C_VEL
LIN {X 0,Y 559.709,Z 504.45,A -85,B 0,C 180,E1 -3071.673,E2 -3071.673} C_VEL
LIN {X 0,Y 559.818,Z 492.957,A -85,B 0,C 180,E1 -3072.185,E2 -3072.185} C_VEL
LIN {X 0,Y 559.963,Z 480.13,A -85,B 0,C 180,E1 -3072.596,E2 -3072.596} C_VEL
LIN {X 0,Y 558.769,Z 471.668,A -85,B 0,C 180,E1 -3072.831,E2 -3072.831} C_VEL
LIN {X 0,Y 558.808,Z 468.454,A -85,B 0,C 180,E1 -3075.314,E2 -3075.314} C_VEL
LIN {X 0,Y 558.774,Z 465.57,A -85,B 0,C 180,E1 -3077.57,E2 -3077.57} C_VEL
LIN {X 0,Y 558.794,Z 462.686,A -85,B 0,C 180,E1 -3079.852,E2 -3079.852} C_VEL
LIN {X 0,Y 558.797,Z 459.864,A -85,B 0,C 180,E1 -3082.168,E2 -3082.168} C_VEL
LIN {X 0,Y 558.849,Z 456.561,A -85,B 0,C 180,E1 -3085.114,E2 -3085.114} C_VEL
LIN {X 0,Y 558.898,Z 454.896,A -85,B 0,C 180,E1 -3086.639,E2 -3086.639} C_VEL
LIN {X 0,Y 558.29,Z 454.271,A -85,B 0,C 180,E1 -3087.237,E2 -3087.237} C_VEL
LIN {X 0,Y 555.484,Z 453.323,A -85,B 0,C 180,E1 -3088.209,E2 -3088.209} C_VEL
LIN {X 0,Y 553.053,Z 452.561,A -85,B 0,C 180,E1 -3088.992,E2 -3088.992} C_VEL
LIN {X 0,Y 551.967,Z 451.934,A -85,B 0,C 180,E1 -3089.595,E2 -3089.595} C_VEL
LIN {X 0,Y 551.858,Z 451.708,A -85,B 0,C 180,E1 -3089.799,E2 -3089.799} C_VEL
LIN {X 0,Y 551.845,Z 448.341,A -85,B 0,C 180,E1 -3092.802,E2 -3092.802} C_VEL
LIN {X 0,Y 551.837,Z 447.89,A -85,B 0,C 180,E1 -3093.205,E2 -3093.205} C_VEL
LIN {X 0,Y 552.03,Z 447.724,A -85,B 0,C 180,E1 -3095.432,E2 -3095.432} C_VEL
LIN {X 0,Y 552.1,Z 447.712,A -85,B 0,C 180,E1 -3097.886,E2 -3097.886} C_VEL
LIN {X 0,Y 552.115,Z 447.71,A -85,B 0,C 180,E1 -3100.481,E2 -3100.481} C_VEL
LIN {X 0,Y 552.125,Z 447.71,A -85,B 0,C 180,E1 -3103.485,E2 -3103.485} C_VEL
LIN {X 0,Y 552.112,Z 447.711,A -85,B 0,C 180,E1 -3106.576,E2 -3106.576} C_VEL
LIN {X 0,Y 552.115,Z 447.713,A -85,B 0,C 180,E1 -3109.519,E2 -3109.519} C_VEL
LIN {X 0,Y 552.098,Z 447.717,A -85,B 0,C 180,E1 -3112.336,E2 -3112.336} C_VEL
LIN {X 0,Y 552.093,Z 447.713,A -85,B 0,C 180,E1 -3115.051,E2 -3115.051} C_VEL
LIN {X 0,Y 552.121,Z 447.71,A -85,B 0,C 180,E1 -3117.681,E2 -3117.681} C_VEL
LIN {X 0,Y 552.113,Z 447.715,A -85,B 0,C 180,E1 -3120.235,E2 -3120.235} C_VEL
LIN {X 0,Y 552.143,Z 447.709,A -85,B 0,C 180,E1 -3123,E2 -3123} C_VEL
LIN {X 0,Y 552.12,Z 447.712,A -85,B 0,C 180,E1 -3125.161,E2 -3125.161} C_VEL
LIN {X 0,Y 552.132,Z 447.709,A -85,B 0,C 180,E1 -3128.337,E2 -3128.337} C_VEL
LIN {X 0,Y 552.157,Z 447.706,A -85,B 0,C 180,E1 -3130.674,E2 -3130.674} C_VEL
LIN {X 0,Y 552.118,Z 447.71,A -85,B 0,C 180,E1 -3133.737,E2 -3133.737} C_VEL
LIN {X 0,Y 552.142,Z 447.71,A -85,B 0,C 180,E1 -3136.004,E2 -3136.004} C_VEL
LIN {X 0,Y 552.169,Z 447.707,A -85,B 0,C 180,E1 -3138.993,E2 -3138.993} C_VEL
LIN {X 0,Y 552.153,Z 447.71,A -85,B 0,C 180,E1 -3141.951,E2 -3141.951} C_VEL
LIN {X 0,Y 552.231,Z 447.698,A -85,B 0,C 180,E1 -3144.889,E2 -3144.889} C_VEL
LIN {X 0,Y 552.23,Z 447.697,A -85,B 0,C 180,E1 -3147.812,E2 -3147.812} C_VEL
LIN {X 0,Y 552.247,Z 447.693,A -85,B 0,C 180,E1 -3150.729,E2 -3150.729} C_VEL
LIN {X 0,Y 552.207,Z 447.703,A -85,B 0,C 180,E1 -3152.918,E2 -3152.918} C_VEL
LIN {X 0,Y 552.195,Z 447.703,A -85,B 0,C 180,E1 -3155.844,E2 -3155.844} C_VEL
LIN {X 0,Y 552.164,Z 447.705,A -85,B 0,C 180,E1 -3158.785,E2 -3158.785} C_VEL
LIN {X 0,Y 552.169,Z 447.704,A -85,B 0,C 180,E1 -3161.75,E2 -3161.75} C_VEL
LIN {X 0,Y 552.142,Z 447.706,A -85,B 0,C 180,E1 -3164.748,E2 -3164.748} C_VEL
LIN {X 0,Y 552.115,Z 447.71,A -85,B 0,C 180,E1 -3167.788,E2 -3167.788} C_VEL
LIN {X 0,Y 552.132,Z 447.713,A -85,B 0,C 180,E1 -3170.101,E2 -3170.101} C_VEL
LIN {X 0,Y 552.098,Z 447.712,A -85,B 0,C 180,E1 -3172.451,E2 -3172.451} C_VEL
LIN {X 0,Y 552.161,Z 447.705,A -85,B 0,C 180,E1 -3175.35,E2 -3175.35} C_VEL
LIN {X 0,Y 552.108,Z 447.714,A -85,B 0,C 180,E1 -3178.098,E2 -3178.098} C_VEL
LIN {X 0,Y 552.109,Z 447.712,A -85,B 0,C 180,E1 -3180.609,E2 -3180.609} C_VEL
LIN {X 0,Y 552.12,Z 447.709,A -85,B 0,C 180,E1 -3183.185,E2 -3183.185} C_VEL
LIN {X 0,Y 552.104,Z 447.715,A -85,B 0,C 180,E1 -3185.842,E2 -3185.842} C_VEL
LIN {X 0,Y 552.126,Z 447.712,A -85,B 0,C 180,E1 -3189.061,E2 -3189.061} C_VEL
LIN {X 0,Y 552.124,Z 447.709,A -85,B 0,C 180,E1 -3191.446,E2 -3191.446} C_VEL
LIN {X 0,Y 552.099,Z 447.713,A -85,B 0,C 180,E1 -3194.531,E2 -3194.531} C_VEL
LIN {X 0,Y 552.135,Z 447.708,A -85,B 0,C 180,E1 -3197.584,E2 -3197.584} C_VEL
LIN {X 0,Y 552.132,Z 447.707,A -85,B 0,C 180,E1 -3200.472,E2 -3200.472} C_VEL
LIN {X 0,Y 552.118,Z 447.711,A -85,B 0,C 180,E1 -3203.315,E2 -3203.315} C_VEL
LIN {X 0,Y 552.131,Z 447.713,A -85,B 0,C 180,E1 -3205.939,E2 -3205.939} C_VEL
LIN {X 0,Y 552.122,Z 447.709,A -85,B 0,C 180,E1 -3208.54,E2 -3208.54} C_VEL
LIN {X 0,Y 552.127,Z 447.709,A -85,B 0,C 180,E1 -3211.438,E2 -3211.438} C_VEL
LIN {X 0,Y 552.132,Z 447.707,A -85,B 0,C 180,E1 -3214.355,E2 -3214.355} C_VEL
LIN {X 0,Y 552.101,Z 447.716,A -85,B 0,C 180,E1 -3216.758,E2 -3216.758} C_VEL
LIN {X 0,Y 552.123,Z 447.709,A -85,B 0,C 180,E1 -3219.12,E2 -3219.12} C_VEL
LIN {X 0,Y 552.125,Z 447.713,A -85,B 0,C 180,E1 -3221.444,E2 -3221.444} C_VEL
LIN {X 0,Y 552.119,Z 447.71,A -85,B 0,C 180,E1 -3223.737,E2 -3223.737} C_VEL
LIN {X 0,Y 552.138,Z 447.71,A -85,B 0,C 180,E1 -3226.004,E2 -3226.004} C_VEL
LIN {X 0,Y 552.164,Z 447.705,A -85,B 0,C 180,E1 -3228.993,E2 -3228.993} C_VEL
LIN {X 0,Y 552.161,Z 447.705,A -85,B 0,C 180,E1 -3231.951,E2 -3231.951} C_VEL
LIN {X 0,Y 552.23,Z 447.695,A -85,B 0,C 180,E1 -3234.889,E2 -3234.889} C_VEL
LIN {X 0,Y 552.222,Z 447.697,A -85,B 0,C 180,E1 -3237.812,E2 -3237.812} C_VEL
LIN {X 0,Y 552.245,Z 447.695,A -85,B 0,C 180,E1 -3240.729,E2 -3240.729} C_VEL
LIN {X 0,Y 552.208,Z 447.699,A -85,B 0,C 180,E1 -3242.918,E2 -3242.918} C_VEL
LIN {X 0,Y 552.2,Z 447.7,A -85,B 0,C 180,E1 -3245.844,E2 -3245.844} C_VEL
LIN {X 0,Y 552.159,Z 447.704,A -85,B 0,C 180,E1 -3248.786,E2 -3248.786} C_VEL
LIN {X 0,Y 552.164,Z 447.704,A -85,B 0,C 180,E1 -3251.75,E2 -3251.75} C_VEL
LIN {X 0,Y 552.138,Z 447.708,A -85,B 0,C 180,E1 -3254.748,E2 -3254.748} C_VEL
LIN {X 0,Y 552.112,Z 447.711,A -85,B 0,C 180,E1 -3257.788,E2 -3257.788} C_VEL
LIN {X 0,Y 552.133,Z 447.709,A -85,B 0,C 180,E1 -3260.101,E2 -3260.101} C_VEL
LIN {X 0,Y 552.095,Z 447.714,A -85,B 0,C 180,E1 -3262.451,E2 -3262.451} C_VEL
LIN {X 0,Y 552.157,Z 447.709,A -85,B 0,C 180,E1 -3265.35,E2 -3265.35} C_VEL
LIN {X 0,Y 552.121,Z 447.713,A -85,B 0,C 180,E1 -3268.098,E2 -3268.098} C_VEL
LIN {X 0,Y 552.104,Z 447.711,A -85,B 0,C 180,E1 -3270.609,E2 -3270.609} C_VEL
LIN {X 0,Y 552.116,Z 447.713,A -85,B 0,C 180,E1 -3273.186,E2 -3273.186} C_VEL
LIN {X 0,Y 552.11,Z 447.713,A -85,B 0,C 180,E1 -3275.842,E2 -3275.842} C_VEL
LIN {X 0,Y 552.122,Z 447.712,A -85,B 0,C 180,E1 -3279.061,E2 -3279.061} C_VEL
LIN {X 0,Y 552.14,Z 447.707,A -85,B 0,C 180,E1 -3281.444,E2 -3281.444} C_VEL
LIN {X 0,Y 552.096,Z 447.714,A -85,B 0,C 180,E1 -3284.532,E2 -3284.532} C_VEL
LIN {X 0,Y 552.13,Z 447.71,A -85,B 0,C 180,E1 -3287.585,E2 -3287.585} C_VEL
LIN {X 0,Y 552.136,Z 447.711,A -85,B 0,C 180,E1 -3290.473,E2 -3290.473} C_VEL
LIN {X 0,Y 552.132,Z 447.769,A -85,B 0,C 180,E1 -3292.512,E2 -3292.512} C_VEL
LIN {X 0,Y 552.927,Z 453.079,A -85,B 0,C 180,E1 -3294.437,E2 -3294.437} C_VEL
LIN {X 0,Y 552.829,Z 460.243,A -85,B 0,C 180,E1 -3296.863,E2 -3296.863} C_VEL
LIN {X 0,Y 552.648,Z 469.448,A -85,B 0,C 180,E1 -3299.855,E2 -3299.855} C_VEL
LIN {X 0,Y 552.473,Z 479.39,A -85,B 0,C 180,E1 -3302.933,E2 -3302.933} C_VEL
LIN {X 0,Y 552.325,Z 489.433,A -85,B 0,C 180,E1 -3305.972,E2 -3305.972} C_VEL
LIN {X 0,Y 552.199,Z 498.889,A -85,B 0,C 180,E1 -3308.732,E2 -3308.732} C_VEL
LIN {X 0,Y 552.085,Z 508.169,A -85,B 0,C 180,E1 -3311.443,E2 -3311.443} C_VEL
LIN {X 0,Y 551.981,Z 518.76,A -85,B 0,C 180,E1 -3314.492,E2 -3314.492} C_VEL
LIN {X 0,Y 551.909,Z 527.531,A -85,B 0,C 180,E1 -3316.984,E2 -3316.984} C_VEL
LIN {X 0,Y 553.097,Z 535.515,A -85,B 0,C 180,E1 -3317.175,E2 -3317.175} C_VEL
LIN {X 0,Y 552.972,Z 547.878,A -85,B 0,C 180,E1 -3317.522,E2 -3317.522} C_VEL
LIN {X 0,Y 552.813,Z 559.509,A -85,B 0,C 180,E1 -3317.985,E2 -3317.985} C_VEL
LIN {X 0,Y 552.633,Z 571.899,A -85,B 0,C 180,E1 -3318.638,E2 -3318.638} C_VEL
LIN {X 0,Y 552.415,Z 582.747,A -85,B 0,C 180,E1 -3319.37,E2 -3319.37} C_VEL
LIN {X 0,Y 552.232,Z 593.601,A -85,B 0,C 180,E1 -3320.292,E2 -3320.292} C_VEL
LIN {X 0,Y 552.079,Z 602.414,A -85,B 0,C 180,E1 -3321.213,E2 -3321.213} C_VEL
LIN {X 0,Y 551.949,Z 611.003,A -85,B 0,C 180,E1 -3322.317,E2 -3322.317} C_VEL
LIN {X 0,Y 551.823,Z 617.869,A -85,B 0,C 180,E1 -3323.418,E2 -3323.418} C_VEL
LIN {X 0,Y 551.804,Z 623.367,A -85,B 0,C 180,E1 -3324.519,E2 -3324.519} C_VEL
LIN {X 0,Y 551.764,Z 627.678,A -85,B 0,C 180,E1 -3325.617,E2 -3325.617} C_VEL
LIN {X 0,Y 551.75,Z 629.958,A -85,B 0,C 180,E1 -3326.349,E2 -3326.349} C_VEL
LIN {X 0,Y 551.723,Z 631.808,A -85,B 0,C 180,E1 -3327.079,E2 -3327.079} C_VEL
LIN {X 0,Y 551.645,Z 634.185,A -85,B 0,C 180,E1 -3328.54,E2 -3328.54} C_VEL
LIN {X 0,Y 551.64,Z 635,A -85,B 0,C 180,E1 -3330,E2 -3330} C_VEL
LIN {X 0,Y 551.645,Z 634.185,A -85,B 0,C 180,E1 -3331.46,E2 -3331.46} C_VEL
LIN {X 0,Y 551.723,Z 631.81,A -85,B 0,C 180,E1 -3332.921,E2 -3332.921} C_VEL
LIN {X 0,Y 551.764,Z 628.895,A -85,B 0,C 180,E1 -3334.017,E2 -3334.017} C_VEL
LIN {X 0,Y 551.724,Z 624.948,A -85,B 0,C 180,E1 -3335.116,E2 -3335.116} C_VEL
LIN {X 0,Y 551.803,Z 619.188,A -85,B 0,C 180,E1 -3336.342,E2 -3336.342} C_VEL
LIN {X 0,Y 551.926,Z 612.235,A -85,B 0,C 180,E1 -3337.5,E2 -3337.5} C_VEL
LIN {X 0,Y 552.082,Z 603.99,A -85,B 0,C 180,E1 -3338.603,E2 -3338.603} C_VEL
LIN {X 0,Y 552.201,Z 595.537,A -85,B 0,C 180,E1 -3339.524,E2 -3339.524} C_VEL
LIN {X 0,Y 552.419,Z 585.093,A -85,B 0,C 180,E1 -3340.445,E2 -3340.445} C_VEL
LIN {X 0,Y 552.59,Z 574.294,A -85,B 0,C 180,E1 -3341.213,E2 -3341.213} C_VEL
LIN {X 0,Y 552.754,Z 563.404,A -85,B 0,C 180,E1 -3341.831,E2 -3341.831} C_VEL
LIN {X 0,Y 552.902,Z 551.758,A -85,B 0,C 180,E1 -3342.34,E2 -3342.34} C_VEL
LIN {X 0,Y 553.063,Z 539.253,A -85,B 0,C 180,E1 -3342.732,E2 -3342.732} C_VEL
LIN {X 0,Y 552.905,Z 533.785,A -85,B 0,C 180,E1 -3342.864,E2 -3342.864} C_VEL
LIN {X 0,Y 551.909,Z 527.529,A -85,B 0,C 180,E1 -3343.017,E2 -3343.017} C_VEL
LIN {X 0,Y 551.996,Z 517.435,A -85,B 0,C 180,E1 -3345.887,E2 -3345.887} C_VEL
LIN {X 0,Y 552.085,Z 506.844,A -85,B 0,C 180,E1 -3348.942,E2 -3348.942} C_VEL
LIN {X 0,Y 552.185,Z 497.337,A -85,B 0,C 180,E1 -3351.702,E2 -3351.702} C_VEL
LIN {X 0,Y 552.304,Z 487.75,A -85,B 0,C 180,E1 -3354.429,E2 -3354.429} C_VEL
LIN {X 0,Y 552.409,Z 478.027,A -85,B 0,C 180,E1 -3357.259,E2 -3357.259} C_VEL
LIN {X 0,Y 552.583,Z 467.311,A -85,B 0,C 180,E1 -3360.58,E2 -3360.58} C_VEL
LIN {X 0,Y 552.751,Z 458.538,A -85,B 0,C 180,E1 -3363.579,E2 -3363.579} C_VEL
LIN {X 0,Y 552.972,Z 452.85,A -85,B 0,C 180,E1 -3365.778,E2 -3365.778} C_VEL
LIN {X 0,Y 552.234,Z 448.353,A -85,B 0,C 180,E1 -3367.904,E2 -3367.904} C_VEL
LIN {X 0,Y 552.126,Z 447.714,A -85,B 0,C 180,E1 -3368.398,E2 -3368.398} C_VEL
LIN {X 0,Y 552.132,Z 447.713,A -85,B 0,C 180,E1 -3371.445,E2 -3371.445} C_VEL
LIN {X 0,Y 552.099,Z 447.716,A -85,B 0,C 180,E1 -3374.532,E2 -3374.532} C_VEL
LIN {X 0,Y 552.135,Z 447.713,A -85,B 0,C 180,E1 -3377.585,E2 -3377.585} C_VEL
LIN {X 0,Y 552.136,Z 447.711,A -85,B 0,C 180,E1 -3380.473,E2 -3380.473} C_VEL
LIN {X 0,Y 552.105,Z 447.717,A -85,B 0,C 180,E1 -3383.318,E2 -3383.318} C_VEL
LIN {X 0,Y 552.026,Z 447.787,A -85,B 0,C 180,E1 -3385.047,E2 -3385.047} C_VEL
LIN {X 0,Y 552.005,Z 450.34,A -85,B 0,C 180,E1 -3387.674,E2 -3387.674} C_VEL
LIN {X 0,Y 551.962,Z 452.88,A -85,B 0,C 180,E1 -3390.226,E2 -3390.226} C_VEL
LIN {X 0,Y 551.86,Z 455.737,A -85,B 0,C 180,E1 -3393.058,E2 -3393.058} C_VEL
LIN {X 0,Y 551.801,Z 458.653,A -85,B 0,C 180,E1 -3395.948,E2 -3395.948} C_VEL
LIN {X 0,Y 551.723,Z 461.953,A -85,B 0,C 180,E1 -3399.104,E2 -3399.104} C_VEL
LIN {X 0,Y 551.67,Z 464.496,A -85,B 0,C 180,E1 -3401.429,E2 -3401.429} C_VEL
LIN {X 0,Y 551.708,Z 467.379,A -85,B 0,C 180,E1 -3403.725,E2 -3403.725} C_VEL
LIN {X 0,Y 551.7,Z 470.261,A -85,B 0,C 180,E1 -3405.993,E2 -3405.993} C_VEL
LIN {X 0,Y 551.674,Z 471.673,A -85,B 0,C 180,E1 -3407.095,E2 -3407.095} C_VEL
LIN {X 0,Y 553.037,Z 480.243,A -85,B 0,C 180,E1 -3407.337,E2 -3407.337} C_VEL
LIN {X 0,Y 552.878,Z 493.017,A -85,B 0,C 180,E1 -3407.753,E2 -3407.753} C_VEL
LIN {X 0,Y 552.718,Z 504.321,A -85,B 0,C 180,E1 -3408.262,E2 -3408.262} C_VEL
LIN {X 0,Y 552.582,Z 515.76,A -85,B 0,C 180,E1 -3408.927,E2 -3408.927} C_VEL
LIN {X 0,Y 552.369,Z 526.859,A -85,B 0,C 180,E1 -3409.739,E2 -3409.739} C_VEL
LIN {X 0,Y 552.174,Z 536.902,A -85,B 0,C 180,E1 -3410.661,E2 -3410.661} C_VEL
LIN {X 0,Y 552.007,Z 546.601,A -85,B 0,C 180,E1 -3411.765,E2 -3411.765} C_VEL
LIN {X 0,Y 551.895,Z 554.46,A -85,B 0,C 180,E1 -3412.886,E2 -3412.886} C_VEL
LIN {X 0,Y 551.868,Z 561.458,A -85,B 0,C 180,E1 -3414.153,E2 -3414.153} C_VEL
LIN {X 0,Y 551.725,Z 566.198,A -85,B 0,C 180,E1 -3415.251,E2 -3415.251} C_VEL
LIN {X 0,Y 551.751,Z 569.83,A -85,B 0,C 180,E1 -3416.349,E2 -3416.349} C_VEL
LIN {X 0,Y 551.724,Z 571.706,A -85,B 0,C 180,E1 -3417.079,E2 -3417.079} C_VEL
LIN {X 0,Y 551.656,Z 573.129,A -85,B 0,C 180,E1 -3417.81,E2 -3417.81} C_VEL
LIN {X 0,Y 551.642,Z 574.757,A -85,B 0,C 180,E1 -3419.27,E2 -3419.27} C_VEL
LIN {X 0,Y 551.641,Z 574.996,A -85,B 0,C 180,E1 -3420,E2 -3420} C_VEL
LIN {X 0,Y 551.642,Z 574.814,A -85,B 0,C 180,E1 -3420.73,E2 -3420.73} C_VEL
LIN {X 0,Y 551.655,Z 573.265,A -85,B 0,C 180,E1 -3422.191,E2 -3422.191} C_VEL
LIN {X 0,Y 551.724,Z 571.904,A -85,B 0,C 180,E1 -3422.921,E2 -3422.921} C_VEL
LIN {X 0,Y 551.764,Z 569.026,A -85,B 0,C 180,E1 -3424.017,E2 -3424.017} C_VEL
LIN {X 0,Y 551.723,Z 565.124,A -85,B 0,C 180,E1 -3425.116,E2 -3425.116} C_VEL
LIN {X 0,Y 551.81,Z 559.397,A -85,B 0,C 180,E1 -3426.349,E2 -3426.349} C_VEL
LIN {X 0,Y 551.926,Z 552.536,A -85,B 0,C 180,E1 -3427.5,E2 -3427.5} C_VEL
LIN {X 0,Y 552.063,Z 544.352,A -85,B 0,C 180,E1 -3428.603,E2 -3428.603} C_VEL
LIN {X 0,Y 552.197,Z 535.984,A -85,B 0,C 180,E1 -3429.524,E2 -3429.524} C_VEL
LIN {X 0,Y 552.402,Z 525.662,A -85,B 0,C 180,E1 -3430.446,E2 -3430.446} C_VEL
LIN {X 0,Y 552.583,Z 513.878,A -85,B 0,C 180,E1 -3431.286,E2 -3431.286} C_VEL
LIN {X 0,Y 552.76,Z 502.438,A -85,B 0,C 180,E1 -3431.924,E2 -3431.924} C_VEL
LIN {X 0,Y 552.93,Z 490.424,A -85,B 0,C 180,E1 -3432.432,E2 -3432.432} C_VEL
LIN {X 0,Y 552.843,Z 478.733,A -85,B 0,C 180,E1 -3432.796,E2 -3432.796} C_VEL
LIN {X 0,Y 551.673,Z 471.668,A -85,B 0,C 180,E1 -3432.999,E2 -3432.999} C_VEL
LIN {X 0,Y 551.722,Z 468.453,A -85,B 0,C 180,E1 -3435.516,E2 -3435.516} C_VEL
LIN {X 0,Y 551.685,Z 465.569,A -85,B 0,C 180,E1 -3437.803,E2 -3437.803} C_VEL
LIN {X 0,Y 551.692,Z 462.734,A -85,B 0,C 180,E1 -3440.118,E2 -3440.118} C_VEL
LIN {X 0,Y 551.728,Z 460.064,A -85,B 0,C 180,E1 -3442.467,E2 -3442.467} C_VEL
LIN {X 0,Y 551.781,Z 456.972,A -85,B 0,C 180,E1 -3445.267,E2 -3445.267} C_VEL
LIN {X 0,Y 551.808,Z 454.638,A -85,B 0,C 180,E1 -3447.291,E2 -3447.291} C_VEL
LIN {X 0,Y 551.858,Z 451.708,A -85,B 0,C 180,E1 -3449.799,E2 -3449.799} C_VEL
LIN {X 0,Y 551.136,Z 451.083,A -85,B 0,C 180,E1 -3450.405,E2 -3450.405} C_VEL
LIN {X 0,Y 548.268,Z 450.226,A -85,B 0,C 180,E1 -3451.39,E2 -3451.39} C_VEL
LIN {X 0,Y 545.88,Z 449.553,A -85,B 0,C 180,E1 -3452.184,E2 -3452.184} C_VEL
LIN {X 0,Y 544.858,Z 448.966,A -85,B 0,C 180,E1 -3452.795,E2 -3452.795} C_VEL
LIN {X 0,Y 544.774,Z 448.743,A -85,B 0,C 180,E1 -3453.002,E2 -3453.002} C_VEL
LIN {X 0,Y 544.996,Z 448.6,A -85,B 0,C 180,E1 -3455.472,E2 -3455.472} C_VEL
LIN {X 0,Y 545.054,Z 448.592,A -85,B 0,C 180,E1 -3458.136,E2 -3458.136} C_VEL
LIN {X 0,Y 545.087,Z 448.586,A -85,B 0,C 180,E1 -3460.473,E2 -3460.473} C_VEL
LIN {X 0,Y 545.084,Z 448.59,A -85,B 0,C 180,E1 -3463.107,E2 -3463.107} C_VEL
LIN {X 0,Y 545.054,Z 448.594,A -85,B 0,C 180,E1 -3466.226,E2 -3466.226} C_VEL
LIN {X 0,Y 545.087,Z 448.587,A -85,B 0,C 180,E1 -3468.886,E2 -3468.886} C_VEL
LIN {X 0,Y 545.088,Z 448.59,A -85,B 0,C 180,E1 -3470.819,E2 -3470.819} C_VEL
LIN {X 0,Y 545.048,Z 448.591,A -85,B 0,C 180,E1 -3473.62,E2 -3473.62} C_VEL
LIN {X 0,Y 545.073,Z 448.587,A -85,B 0,C 180,E1 -3476.328,E2 -3476.328} C_VEL
LIN {X 0,Y 545.07,Z 448.589,A -85,B 0,C 180,E1 -3478.952,E2 -3478.952} C_VEL
LIN {X 0,Y 545.089,Z 448.587,A -85,B 0,C 180,E1 -3481.507,E2 -3481.507} C_VEL
LIN {X 0,Y 545.102,Z 448.585,A -85,B 0,C 180,E1 -3484.491,E2 -3484.491} C_VEL
LIN {X 0,Y 545.044,Z 448.59,A -85,B 0,C 180,E1 -3487.242,E2 -3487.242} C_VEL
LIN {X 0,Y 545.123,Z 448.581,A -85,B 0,C 180,E1 -3490.415,E2 -3490.415} C_VEL
LIN {X 0,Y 545.069,Z 448.587,A -85,B 0,C 180,E1 -3493.521,E2 -3493.521} C_VEL
LIN {X 0,Y 545.102,Z 448.589,A -85,B 0,C 180,E1 -3495.82,E2 -3495.82} C_VEL
LIN {X 0,Y 545.125,Z 448.585,A -85,B 0,C 180,E1 -3498.849,E2 -3498.849} C_VEL
LIN {X 0,Y 545.102,Z 448.587,A -85,B 0,C 180,E1 -3501.846,E2 -3501.846} C_VEL
LIN {X 0,Y 545.175,Z 448.575,A -85,B 0,C 180,E1 -3504.08,E2 -3504.08} C_VEL
LIN {X 0,Y 545.174,Z 448.576,A -85,B 0,C 180,E1 -3507.044,E2 -3507.044} C_VEL
LIN {X 0,Y 545.209,Z 448.574,A -85,B 0,C 180,E1 -3510,E2 -3510} C_VEL
LIN {X 0,Y 545.174,Z 448.579,A -85,B 0,C 180,E1 -3512.956,E2 -3512.956} C_VEL
LIN {X 0,Y 545.165,Z 448.579,A -85,B 0,C 180,E1 -3515.919,E2 -3515.919} C_VEL
LIN {X 0,Y 545.123,Z 448.583,A -85,B 0,C 180,E1 -3518.9,E2 -3518.9} C_VEL
LIN {X 0,Y 545.141,Z 448.58,A -85,B 0,C 180,E1 -3521.904,E2 -3521.904} C_VEL
LIN {X 0,Y 545.091,Z 448.585,A -85,B 0,C 180,E1 -3524.943,E2 -3524.943} C_VEL
LIN {X 0,Y 545.083,Z 448.587,A -85,B 0,C 180,E1 -3528.026,E2 -3528.026} C_VEL
LIN {X 0,Y 545.098,Z 448.586,A -85,B 0,C 180,E1 -3530.372,E2 -3530.372} C_VEL
LIN {X 0,Y 545.087,Z 448.588,A -85,B 0,C 180,E1 -3533.559,E2 -3533.559} C_VEL
LIN {X 0,Y 545.083,Z 448.588,A -85,B 0,C 180,E1 -3536,E2 -3536} C_VEL
LIN {X 0,Y 545.094,Z 448.584,A -85,B 0,C 180,E1 -3538.748,E2 -3538.748} C_VEL
LIN {X 0,Y 545.062,Z 448.589,A -85,B 0,C 180,E1 -3541.678,E2 -3541.678} C_VEL
LIN {X 0,Y 545.082,Z 448.586,A -85,B 0,C 180,E1 -3544.563,E2 -3544.563} C_VEL
LIN {X 0,Y 545.042,Z 448.596,A -85,B 0,C 180,E1 -3547.303,E2 -3547.303} C_VEL
LIN {X 0,Y 545.069,Z 448.591,A -85,B 0,C 180,E1 -3550.142,E2 -3550.142} C_VEL
LIN {X 0,Y 545.082,Z 448.587,A -85,B 0,C 180,E1 -3553.106,E2 -3553.106} C_VEL
LIN {X 0,Y 545.069,Z 448.59,A -85,B 0,C 180,E1 -3556.224,E2 -3556.224} C_VEL
LIN {X 0,Y 545.091,Z 448.584,A -85,B 0,C 180,E1 -3558.886,E2 -3558.886} C_VEL
LIN {X 0,Y 545.055,Z 448.59,A -85,B 0,C 180,E1 -3561.762,E2 -3561.762} C_VEL
LIN {X 0,Y 545.06,Z 448.592,A -85,B 0,C 180,E1 -3564.533,E2 -3564.533} C_VEL
LIN {X 0,Y 545.083,Z 448.587,A -85,B 0,C 180,E1 -3567.212,E2 -3567.212} C_VEL
LIN {X 0,Y 545.068,Z 448.588,A -85,B 0,C 180,E1 -3569.81,E2 -3569.81} C_VEL
LIN {X 0,Y 545.094,Z 448.588,A -85,B 0,C 180,E1 -3572.344,E2 -3572.344} C_VEL
LIN {X 0,Y 545.12,Z 448.581,A -85,B 0,C 180,E1 -3574.82,E2 -3574.82} C_VEL
LIN {X 0,Y 545.041,Z 448.593,A -85,B 0,C 180,E1 -3577.242,E2 -3577.242} C_VEL
LIN {X 0,Y 545.123,Z 448.581,A -85,B 0,C 180,E1 -3580.415,E2 -3580.415} C_VEL
LIN {X 0,Y 545.076,Z 448.588,A -85,B 0,C 180,E1 -3583.521,E2 -3583.521} C_VEL
LIN {X 0,Y 545.098,Z 448.586,A -85,B 0,C 180,E1 -3585.82,E2 -3585.82} C_VEL
LIN {X 0,Y 545.12,Z 448.581,A -85,B 0,C 180,E1 -3588.849,E2 -3588.849} C_VEL
LIN {X 0,Y 545.132,Z 448.58,A -85,B 0,C 180,E1 -3591.847,E2 -3591.847} C_VEL
LIN {X 0,Y 545.206,Z 448.57,A -85,B 0,C 180,E1 -3594.823,E2 -3594.823} C_VEL
LIN {X 0,Y 545.194,Z 448.572,A -85,B 0,C 180,E1 -3597.783,E2 -3597.783} C_VEL
LIN {X 0,Y 545.215,Z 448.57,A -85,B 0,C 180,E1 -3600.738,E2 -3600.738} C_VEL
LIN {X 0,Y 545.174,Z 448.575,A -85,B 0,C 180,E1 -3602.956,E2 -3602.956} C_VEL
LIN {X 0,Y 545.171,Z 448.576,A -85,B 0,C 180,E1 -3605.919,E2 -3605.919} C_VEL
LIN {X 0,Y 545.118,Z 448.581,A -85,B 0,C 180,E1 -3608.9,E2 -3608.9} C_VEL
LIN {X 0,Y 545.136,Z 448.579,A -85,B 0,C 180,E1 -3611.904,E2 -3611.904} C_VEL
LIN {X 0,Y 545.087,Z 448.586,A -85,B 0,C 180,E1 -3614.943,E2 -3614.943} C_VEL
LIN {X 0,Y 545.08,Z 448.586,A -85,B 0,C 180,E1 -3618.026,E2 -3618.026} C_VEL
LIN {X 0,Y 545.097,Z 448.588,A -85,B 0,C 180,E1 -3620.372,E2 -3620.372} C_VEL
LIN {X 0,Y 545.089,Z 448.59,A -85,B 0,C 180,E1 -3623.559,E2 -3623.559} C_VEL
LIN {X 0,Y 545.081,Z 448.586,A -85,B 0,C 180,E1 -3626,E2 -3626} C_VEL
LIN {X 0,Y 545.09,Z 448.586,A -85,B 0,C 180,E1 -3628.748,E2 -3628.748} C_VEL
LIN {X 0,Y 545.058,Z 448.591,A -85,B 0,C 180,E1 -3631.679,E2 -3631.679} C_VEL
LIN {X 0,Y 545.079,Z 448.591,A -85,B 0,C 180,E1 -3634.563,E2 -3634.563} C_VEL
LIN {X 0,Y 545.04,Z 448.593,A -85,B 0,C 180,E1 -3637.304,E2 -3637.304} C_VEL
LIN {X 0,Y 545.067,Z 448.587,A -85,B 0,C 180,E1 -3640.143,E2 -3640.143} C_VEL
LIN {X 0,Y 545.088,Z 448.585,A -85,B 0,C 180,E1 -3643.106,E2 -3643.106} C_VEL
LIN {X 0,Y 545.05,Z 448.592,A -85,B 0,C 180,E1 -3646.226,E2 -3646.226} C_VEL
LIN {X 0,Y 545.093,Z 448.589,A -85,B 0,C 180,E1 -3648.887,E2 -3648.887} C_VEL
LIN {X 0,Y 545.055,Z 448.593,A -85,B 0,C 180,E1 -3651.763,E2 -3651.763} C_VEL
LIN {X 0,Y 545.09,Z 448.723,A -85,B 0,C 180,E1 -3652.293,E2 -3652.293} C_VEL
LIN {X 0,Y 545.958,Z 453.84,A -85,B 0,C 180,E1 -3654.192,E2 -3654.192} C_VEL
LIN {X 0,Y 545.938,Z 460.192,A -85,B 0,C 180,E1 -3656.389,E2 -3656.389} C_VEL
LIN {X 0,Y 545.683,Z 469.156,A -85,B 0,C 180,E1 -3659.362,E2 -3659.362} C_VEL
LIN {X 0,Y 545.517,Z 478.617,A -85,B 0,C 180,E1 -3662.368,E2 -3662.368} C_VEL
LIN {X 0,Y 545.304,Z 489.275,A -85,B 0,C 180,E1 -3665.643,E2 -3665.643} C_VEL
LIN {X 0,Y 545.153,Z 498.84,A -85,B 0,C 180,E1 -3668.499,E2 -3668.499} C_VEL
LIN {X 0,Y 545.029,Z 509.492,A -85,B 0,C 180,E1 -3671.584,E2 -3671.584} C_VEL
LIN {X 0,Y 544.928,Z 520.084,A -85,B 0,C 180,E1 -3674.669,E2 -3674.669} C_VEL
LIN {X 0,Y 544.825,Z 527.531,A -85,B 0,C 180,E1 -3676.811,E2 -3676.811} C_VEL
LIN {X 0,Y 546.148,Z 536.526,A -85,B 0,C 180,E1 -3677.033,E2 -3677.033} C_VEL
LIN {X 0,Y 546.001,Z 549.178,A -85,B 0,C 180,E1 -3677.408,E2 -3677.408} C_VEL
LIN {X 0,Y 545.847,Z 561.494,A -85,B 0,C 180,E1 -3677.923,E2 -3677.923} C_VEL
LIN {X 0,Y 545.64,Z 573.341,A -85,B 0,C 180,E1 -3678.579,E2 -3678.579} C_VEL
LIN {X 0,Y 545.409,Z 585.096,A -85,B 0,C 180,E1 -3679.419,E2 -3679.419} C_VEL
LIN {X 0,Y 545.165,Z 595.54,A -85,B 0,C 180,E1 -3680.352,E2 -3680.352} C_VEL
LIN {X 0,Y 545.029,Z 603.992,A -85,B 0,C 180,E1 -3681.286,E2 -3681.286} C_VEL
LIN {X 0,Y 544.859,Z 612.237,A -85,B 0,C 180,E1 -3682.403,E2 -3682.403} C_VEL
LIN {X 0,Y 544.733,Z 619.616,A -85,B 0,C 180,E1 -3683.655,E2 -3683.655} C_VEL
LIN {X 0,Y 544.654,Z 624.95,A -85,B 0,C 180,E1 -3684.818,E2 -3684.818} C_VEL
LIN {X 0,Y 544.683,Z 628.895,A -85,B 0,C 180,E1 -3685.931,E2 -3685.931} C_VEL
LIN {X 0,Y 544.65,Z 631.808,A -85,B 0,C 180,E1 -3687.042,E2 -3687.042} C_VEL
LIN {X 0,Y 544.546,Z 634.184,A -85,B 0,C 180,E1 -3688.521,E2 -3688.521} C_VEL
LIN {X 0,Y 544.541,Z 635,A -85,B 0,C 180,E1 -3690,E2 -3690} C_VEL
LIN {X 0,Y 544.546,Z 634.185,A -85,B 0,C 180,E1 -3691.479,E2 -3691.479} C_VEL
LIN {X 0,Y 544.65,Z 631.81,A -85,B 0,C 180,E1 -3692.959,E2 -3692.959} C_VEL
LIN {X 0,Y 544.683,Z 628.895,A -85,B 0,C 180,E1 -3694.07,E2 -3694.07} C_VEL
LIN {X 0,Y 544.654,Z 624.948,A -85,B 0,C 180,E1 -3695.182,E2 -3695.182} C_VEL
LIN {X 0,Y 544.739,Z 619.703,A -85,B 0,C 180,E1 -3696.328,E2 -3696.328} C_VEL
LIN {X 0,Y 544.836,Z 613.466,A -85,B 0,C 180,E1 -3697.412,E2 -3697.412} C_VEL
LIN {X 0,Y 545.007,Z 605.476,A -85,B 0,C 180,E1 -3698.528,E2 -3698.528} C_VEL
LIN {X 0,Y 545.142,Z 597.332,A -85,B 0,C 180,E1 -3699.461,E2 -3699.461} C_VEL
LIN {X 0,Y 545.365,Z 587.397,A -85,B 0,C 180,E1 -3700.394,E2 -3700.394} C_VEL
LIN {X 0,Y 545.561,Z 576.589,A -85,B 0,C 180,E1 -3701.208,E2 -3701.208} C_VEL
LIN {X 0,Y 545.742,Z 565.17,A -85,B 0,C 180,E1 -3701.891,E2 -3701.891} C_VEL
LIN {X 0,Y 545.94,Z 552.97,A -85,B 0,C 180,E1 -3702.452,E2 -3702.452} C_VEL
LIN {X 0,Y 546.125,Z 540.167,A -85,B 0,C 180,E1 -3702.873,E2 -3702.873} C_VEL
LIN {X 0,Y 545.848,Z 533.656,A -85,B 0,C 180,E1 -3703.036,E2 -3703.036} C_VEL
LIN {X 0,Y 544.825,Z 527.529,A -85,B 0,C 180,E1 -3703.189,E2 -3703.189} C_VEL
LIN {X 0,Y 544.939,Z 517.435,A -85,B 0,C 180,E1 -3706.098,E2 -3706.098} C_VEL
LIN {X 0,Y 545.068,Z 506.836,A -85,B 0,C 180,E1 -3709.196,E2 -3709.196} C_VEL
LIN {X 0,Y 545.17,Z 495.599,A -85,B 0,C 180,E1 -3712.352,E2 -3712.352} C_VEL
LIN {X 0,Y 545.297,Z 484.688,A -85,B 0,C 180,E1 -3715.553,E2 -3715.553} C_VEL
LIN {X 0,Y 545.37,Z 476.374,A -85,B 0,C 180,E1 -3718.058,E2 -3718.058} C_VEL
LIN {X 0,Y 545.586,Z 468.315,A -85,B 0,C 180,E1 -3720.632,E2 -3720.632} C_VEL
LIN {X 0,Y 545.782,Z 459.773,A -85,B 0,C 180,E1 -3723.622,E2 -3723.622} C_VEL
LIN {X 0,Y 546.03,Z 454.229,A -85,B 0,C 180,E1 -3725.818,E2 -3725.818} C_VEL
LIN {X 0,Y 545.219,Z 449.355,A -85,B 0,C 180,E1 -3728.224,E2 -3728.224} C_VEL
LIN {X 0,Y 545.098,Z 448.59,A -85,B 0,C 180,E1 -3728.706,E2 -3728.706} C_VEL
LIN {X 0,Y 545.089,Z 448.59,A -85,B 0,C 180,E1 -3731.599,E2 -3731.599} C_VEL
LIN {X 0,Y 545.062,Z 448.593,A -85,B 0,C 180,E1 -3734.129,E2 -3734.129} C_VEL
LIN {X 0,Y 545.09,Z 448.588,A -85,B 0,C 180,E1 -3736.894,E2 -3736.894} C_VEL
LIN {X 0,Y 545.075,Z 448.592,A -85,B 0,C 180,E1 -3739.858,E2 -3739.858} C_VEL
LIN {X 0,Y 545.071,Z 448.592,A -85,B 0,C 180,E1 -3743.074,E2 -3743.074} C_VEL
LIN {X 0,Y 544.995,Z 448.603,A -85,B 0,C 180,E1 -3744.528,E2 -3744.528} C_VEL
LIN {X 0,Y 544.971,Z 449.932,A -85,B 0,C 180,E1 -3746.321,E2 -3746.321} C_VEL
LIN {X 0,Y 544.922,Z 452.461,A -85,B 0,C 180,E1 -3748.943,E2 -3748.943} C_VEL
LIN {X 0,Y 544.853,Z 454.96,A -85,B 0,C 180,E1 -3751.493,E2 -3751.493} C_VEL
LIN {X 0,Y 544.783,Z 458.026,A -85,B 0,C 180,E1 -3754.561,E2 -3754.561} C_VEL
LIN {X 0,Y 544.702,Z 460.745,A -85,B 0,C 180,E1 -3757.227,E2 -3757.227} C_VEL
LIN {X 0,Y 544.673,Z 463.231,A -85,B 0,C 180,E1 -3759.611,E2 -3759.611} C_VEL
LIN {X 0,Y 544.616,Z 466.454,A -85,B 0,C 180,E1 -3762.734,E2 -3762.734} C_VEL
LIN {X 0,Y 544.636,Z 469.777,A -85,B 0,C 180,E1 -3765.422,E2 -3765.422} C_VEL
LIN {X 0,Y 544.593,Z 471.673,A -85,B 0,C 180,E1 -3766.924,E2 -3766.924} C_VEL
LIN {X 0,Y 546.125,Z 481.176,A -85,B 0,C 180,E1 -3767.198,E2 -3767.198} C_VEL
LIN {X 0,Y 545.952,Z 494.159,A -85,B 0,C 180,E1 -3767.643,E2 -3767.643} C_VEL
LIN {X 0,Y 545.729,Z 506.35,A -85,B 0,C 180,E1 -3768.217,E2 -3768.217} C_VEL
LIN {X 0,Y 545.527,Z 518.289,A -85,B 0,C 180,E1 -3768.952,E2 -3768.952} C_VEL
LIN {X 0,Y 545.287,Z 529.025,A -85,B 0,C 180,E1 -3769.792,E2 -3769.792} C_VEL
LIN {X 0,Y 545.122,Z 538.687,A -85,B 0,C 180,E1 -3770.726,E2 -3770.726} C_VEL
LIN {X 0,Y 544.975,Z 546.605,A -85,B 0,C 180,E1 -3771.658,E2 -3771.658} C_VEL
LIN {X 0,Y 544.829,Z 554.352,A -85,B 0,C 180,E1 -3772.775,E2 -3772.775} C_VEL
LIN {X 0,Y 544.778,Z 561.461,A -85,B 0,C 180,E1 -3774.076,E2 -3774.076} C_VEL
LIN {X 0,Y 544.629,Z 566.2,A -85,B 0,C 180,E1 -3775.189,E2 -3775.189} C_VEL
LIN {X 0,Y 544.669,Z 569.832,A -85,B 0,C 180,E1 -3776.301,E2 -3776.301} C_VEL
LIN {X 0,Y 544.651,Z 571.708,A -85,B 0,C 180,E1 -3777.042,E2 -3777.042} C_VEL
LIN {X 0,Y 544.57,Z 573.129,A -85,B 0,C 180,E1 -3777.781,E2 -3777.781} C_VEL
LIN {X 0,Y 544.542,Z 574.758,A -85,B 0,C 180,E1 -3779.261,E2 -3779.261} C_VEL
LIN {X 0,Y 544.541,Z 574.996,A -85,B 0,C 180,E1 -3780,E2 -3780} C_VEL
LIN {X 0,Y 544.542,Z 574.814,A -85,B 0,C 180,E1 -3780.74,E2 -3780.74} C_VEL
LIN {X 0,Y 544.57,Z 573.263,A -85,B 0,C 180,E1 -3782.219,E2 -3782.219} C_VEL
LIN {X 0,Y 544.651,Z 571.902,A -85,B 0,C 180,E1 -3782.959,E2 -3782.959} C_VEL
LIN {X 0,Y 544.684,Z 569.024,A -85,B 0,C 180,E1 -3784.07,E2 -3784.07} C_VEL
LIN {X 0,Y 544.653,Z 565.121,A -85,B 0,C 180,E1 -3785.183,E2 -3785.183} C_VEL
LIN {X 0,Y 544.724,Z 559.9,A -85,B 0,C 180,E1 -3786.334,E2 -3786.334} C_VEL
LIN {X 0,Y 544.859,Z 552.532,A -85,B 0,C 180,E1 -3787.598,E2 -3787.598} C_VEL
LIN {X 0,Y 544.999,Z 544.348,A -85,B 0,C 180,E1 -3788.715,E2 -3788.715} C_VEL
LIN {X 0,Y 545.16,Z 535.978,A -85,B 0,C 180,E1 -3789.648,E2 -3789.648} C_VEL
LIN {X 0,Y 545.379,Z 525.653,A -85,B 0,C 180,E1 -3790.582,E2 -3790.582} C_VEL
LIN {X 0,Y 545.603,Z 514.266,A -85,B 0,C 180,E1 -3791.406,E2 -3791.406} C_VEL
LIN {X 0,Y 545.804,Z 502.427,A -85,B 0,C 180,E1 -3792.078,E2 -3792.078} C_VEL
LIN {X 0,Y 545.991,Z 490.406,A -85,B 0,C 180,E1 -3792.593,E2 -3792.593} C_VEL
LIN {X 0,Y 546.01,Z 480.083,A -85,B 0,C 180,E1 -3792.923,E2 -3792.923} C_VEL
LIN {X 0,Y 544.585,Z 471.667,A -85,B 0,C 180,E1 -3793.171,E2 -3793.171} C_VEL
LIN {X 0,Y 544.626,Z 468.453,A -85,B 0,C 180,E1 -3795.723,E2 -3795.723} C_VEL
LIN {X 0,Y 544.607,Z 465.623,A -85,B 0,C 180,E1 -3798.042,E2 -3798.042} C_VEL
LIN {X 0,Y 544.622,Z 462.931,A -85,B 0,C 180,E1 -3800.391,E2 -3800.391} C_VEL
LIN {X 0,Y 544.644,Z 460.264,A -85,B 0,C 180,E1 -3802.775,E2 -3802.775} C_VEL
LIN {X 0,Y 544.73,Z 457.35,A -85,B 0,C 180,E1 -3805.427,E2 -3805.427} C_VEL
LIN {X 0,Y 544.728,Z 454.697,A -85,B 0,C 180,E1 -3807.676,E2 -3807.676} C_VEL
LIN {X 0,Y 544.758,Z 451.822,A -85,B 0,C 180,E1 -3810.209,E2 -3810.209} C_VEL
LIN {X 0,Y 544.774,Z 448.743,A -85,B 0,C 180,E1 -3813.002,E2 -3813.002} C_VEL
LIN {X 0,Y 544.465,Z 448.667,A -85,B 0,C 180,E1 -3813.413,E2 -3813.413} C_VEL
LIN {X 0,Y 542.589,Z 448.901,A -85,B 0,C 180,E1 -3814.223,E2 -3814.223} C_VEL
LIN {X 0,Y 539.021,Z 449.389,A -85,B 0,C 180,E1 -3815.433,E2 -3815.433} C_VEL
LIN {X 0,Y 538.037,Z 449.468,A -85,B 0,C 180,E1 -3816.058,E2 -3816.058} C_VEL
LIN {X 0,Y 537.966,Z 449.472,A -85,B 0,C 180,E1 -3816.269,E2 -3816.269} C_VEL
LIN {X 0,Y 538.016,Z 449.466,A -85,B 0,C 180,E1 -3818.831,E2 -3818.831} C_VEL
LIN {X 0,Y 538.043,Z 449.466,A -85,B 0,C 180,E1 -3821.773,E2 -3821.773} C_VEL
LIN {X 0,Y 538.013,Z 449.469,A -85,B 0,C 180,E1 -3824.862,E2 -3824.862} C_VEL
LIN {X 0,Y 538.024,Z 449.466,A -85,B 0,C 180,E1 -3827.214,E2 -3827.214} C_VEL
LIN {X 0,Y 538.031,Z 449.465,A -85,B 0,C 180,E1 -3830.203,E2 -3830.203} C_VEL
LIN {X 0,Y 538.03,Z 449.464,A -85,B 0,C 180,E1 -3833.067,E2 -3833.067} C_VEL
LIN {X 0,Y 538.026,Z 449.468,A -85,B 0,C 180,E1 -3835.827,E2 -3835.827} C_VEL
LIN {X 0,Y 538.014,Z 449.471,A -85,B 0,C 180,E1 -3838.499,E2 -3838.499} C_VEL
LIN {X 0,Y 538.025,Z 449.465,A -85,B 0,C 180,E1 -3841.098,E2 -3841.098} C_VEL
LIN {X 0,Y 538.048,Z 449.465,A -85,B 0,C 180,E1 -3843.633,E2 -3843.633} C_VEL
LIN {X 0,Y 538.013,Z 449.469,A -85,B 0,C 180,E1 -3846.122,E2 -3846.122} C_VEL
LIN {X 0,Y 538.044,Z 449.466,A -85,B 0,C 180,E1 -3849.349,E2 -3849.349} C_VEL
LIN {X 0,Y 538.061,Z 449.465,A -85,B 0,C 180,E1 -3852.517,E2 -3852.517} C_VEL
LIN {X 0,Y 538.071,Z 449.462,A -85,B 0,C 180,E1 -3855.631,E2 -3855.631} C_VEL
LIN {X 0,Y 538.084,Z 449.461,A -85,B 0,C 180,E1 -3858.701,E2 -3858.701} C_VEL
LIN {X 0,Y 538.066,Z 449.462,A -85,B 0,C 180,E1 -3861.739,E2 -3861.739} C_VEL
LIN {X 0,Y 538.128,Z 449.454,A -85,B 0,C 180,E1 -3864.003,E2 -3864.003} C_VEL
LIN {X 0,Y 538.141,Z 449.453,A -85,B 0,C 180,E1 -3867.005,E2 -3867.005} C_VEL
LIN {X 0,Y 538.18,Z 449.449,A -85,B 0,C 180,E1 -3870,E2 -3870} C_VEL
LIN {X 0,Y 538.141,Z 449.455,A -85,B 0,C 180,E1 -3872.994,E2 -3872.994} C_VEL
LIN {X 0,Y 538.117,Z 449.458,A -85,B 0,C 180,E1 -3875.997,E2 -3875.997} C_VEL
LIN {X 0,Y 538.074,Z 449.463,A -85,B 0,C 180,E1 -3879.017,E2 -3879.017} C_VEL
LIN {X 0,Y 538.089,Z 449.46,A -85,B 0,C 180,E1 -3882.062,E2 -3882.062} C_VEL
LIN {X 0,Y 538.05,Z 449.464,A -85,B 0,C 180,E1 -3885.143,E2 -3885.143} C_VEL
LIN {X 0,Y 538.035,Z 449.467,A -85,B 0,C 180,E1 -3888.27,E2 -3888.27} C_VEL
LIN {X 0,Y 538.043,Z 449.462,A -85,B 0,C 180,E1 -3890.651,E2 -3890.651} C_VEL
LIN {X 0,Y 538.01,Z 449.467,A -85,B 0,C 180,E1 -3893.888,E2 -3893.888} C_VEL
LIN {X 0,Y 538.045,Z 449.467,A -85,B 0,C 180,E1 -3896.366,E2 -3896.366} C_VEL
LIN {X 0,Y 538.035,Z 449.464,A -85,B 0,C 180,E1 -3898.933,E2 -3898.933} C_VEL
LIN {X 0,Y 538.015,Z 449.467,A -85,B 0,C 180,E1 -3901.887,E2 -3901.887} C_VEL
LIN {X 0,Y 538.032,Z 449.464,A -85,B 0,C 180,E1 -3904.62,E2 -3904.62} C_VEL
LIN {X 0,Y 538.01,Z 449.471,A -85,B 0,C 180,E1 -3907.17,E2 -3907.17} C_VEL
LIN {X 0,Y 538.026,Z 449.466,A -85,B 0,C 180,E1 -3909.797,E2 -3909.797} C_VEL
LIN {X 0,Y 538.022,Z 449.465,A -85,B 0,C 180,E1 -3912.786,E2 -3912.786} C_VEL
LIN {X 0,Y 538.036,Z 449.469,A -85,B 0,C 180,E1 -3915.14,E2 -3915.14} C_VEL
LIN {X 0,Y 538.04,Z 449.467,A -85,B 0,C 180,E1 -3918.227,E2 -3918.227} C_VEL
LIN {X 0,Y 538.015,Z 449.47,A -85,B 0,C 180,E1 -3921.169,E2 -3921.169} C_VEL
LIN {X 0,Y 538.03,Z 449.467,A -85,B 0,C 180,E1 -3924.083,E2 -3924.083} C_VEL
LIN {X 0,Y 538.033,Z 449.463,A -85,B 0,C 180,E1 -3926.727,E2 -3926.727} C_VEL
LIN {X 0,Y 538.029,Z 449.466,A -85,B 0,C 180,E1 -3929.556,E2 -3929.556} C_VEL
LIN {X 0,Y 538.048,Z 449.465,A -85,B 0,C 180,E1 -3931.95,E2 -3931.95} C_VEL
LIN {X 0,Y 538.073,Z 449.458,A -85,B 0,C 180,E1 -3934.467,E2 -3934.467} C_VEL
LIN {X 0,Y 537.996,Z 449.469,A -85,B 0,C 180,E1 -3937.738,E2 -3937.738} C_VEL
LIN {X 0,Y 538.082,Z 449.461,A -85,B 0,C 180,E1 -3940.148,E2 -3940.148} C_VEL
LIN {X 0,Y 538.027,Z 449.468,A -85,B 0,C 180,E1 -3943.299,E2 -3943.299} C_VEL
LIN {X 0,Y 538.066,Z 449.461,A -85,B 0,C 180,E1 -3945.63,E2 -3945.63} C_VEL
LIN {X 0,Y 538.079,Z 449.457,A -85,B 0,C 180,E1 -3948.701,E2 -3948.701} C_VEL
LIN {X 0,Y 538.089,Z 449.457,A -85,B 0,C 180,E1 -3951.739,E2 -3951.739} C_VEL
LIN {X 0,Y 538.163,Z 449.447,A -85,B 0,C 180,E1 -3954.755,E2 -3954.755} C_VEL
LIN {X 0,Y 538.167,Z 449.448,A -85,B 0,C 180,E1 -3957.755,E2 -3957.755} C_VEL
LIN {X 0,Y 538.185,Z 449.446,A -85,B 0,C 180,E1 -3960.748,E2 -3960.748} C_VEL
LIN {X 0,Y 538.14,Z 449.451,A -85,B 0,C 180,E1 -3962.994,E2 -3962.994} C_VEL
LIN {X 0,Y 538.125,Z 449.454,A -85,B 0,C 180,E1 -3965.997,E2 -3965.997} C_VEL
LIN {X 0,Y 538.069,Z 449.46,A -85,B 0,C 180,E1 -3969.018,E2 -3969.018} C_VEL
LIN {X 0,Y 538.085,Z 449.458,A -85,B 0,C 180,E1 -3972.062,E2 -3972.062} C_VEL
LIN {X 0,Y 538.047,Z 449.463,A -85,B 0,C 180,E1 -3975.144,E2 -3975.144} C_VEL
LIN {X 0,Y 538.033,Z 449.464,A -85,B 0,C 180,E1 -3978.27,E2 -3978.27} C_VEL
LIN {X 0,Y 538.041,Z 449.468,A -85,B 0,C 180,E1 -3980.651,E2 -3980.651} C_VEL
LIN {X 0,Y 538.026,Z 449.467,A -85,B 0,C 180,E1 -3983.887,E2 -3983.887} C_VEL
LIN {X 0,Y 538.043,Z 449.464,A -85,B 0,C 180,E1 -3986.367,E2 -3986.367} C_VEL
LIN {X 0,Y 538.032,Z 449.465,A -85,B 0,C 180,E1 -3988.934,E2 -3988.934} C_VEL
LIN {X 0,Y 538.011,Z 449.467,A -85,B 0,C 180,E1 -3991.887,E2 -3991.887} C_VEL
LIN {X 0,Y 538.029,Z 449.469,A -85,B 0,C 180,E1 -3994.62,E2 -3994.62} C_VEL
LIN {X 0,Y 538.009,Z 449.468,A -85,B 0,C 180,E1 -3997.171,E2 -3997.171} C_VEL
LIN {X 0,Y 538.024,Z 449.465,A -85,B 0,C 180,E1 -3999.797,E2 -3999.797} C_VEL
LIN {X 0,Y 538.025,Z 449.467,A -85,B 0,C 180,E1 -4002.785,E2 -4002.785} C_VEL
LIN {X 0,Y 538.008,Z 449.471,A -85,B 0,C 180,E1 -4005.138,E2 -4005.138} C_VEL
LIN {X 0,Y 538.036,Z 449.467,A -85,B 0,C 180,E1 -4008.227,E2 -4008.227} C_VEL
LIN {X 0,Y 538.017,Z 449.468,A -85,B 0,C 180,E1 -4011.17,E2 -4011.17} C_VEL
LIN {X 0,Y 538.035,Z 449.477,A -85,B 0,C 180,E1 -4011.998,E2 -4011.998} C_VEL
LIN {X 0,Y 538.963,Z 454.968,A -85,B 0,C 180,E1 -4014.07,E2 -4014.07} C_VEL
LIN {X 0,Y 538.991,Z 460.141,A -85,B 0,C 180,E1 -4015.897,E2 -4015.897} C_VEL
LIN {X 0,Y 538.718,Z 469.266,A -85,B 0,C 180,E1 -4018.982,E2 -4018.982} C_VEL
LIN {X 0,Y 538.492,Z 478.477,A -85,B 0,C 180,E1 -4021.976,E2 -4021.976} C_VEL
LIN {X 0,Y 538.297,Z 487.786,A -85,B 0,C 180,E1 -4024.893,E2 -4024.893} C_VEL
LIN {X 0,Y 538.114,Z 497.985,A -85,B 0,C 180,E1 -4028.017,E2 -4028.017} C_VEL
LIN {X 0,Y 537.983,Z 507.962,A -85,B 0,C 180,E1 -4030.938,E2 -4030.938} C_VEL
LIN {X 0,Y 537.879,Z 517.436,A -85,B 0,C 180,E1 -4033.685,E2 -4033.685} C_VEL
LIN {X 0,Y 537.772,Z 526.703,A -85,B 0,C 180,E1 -4036.395,E2 -4036.395} C_VEL
LIN {X 0,Y 537.764,Z 527.572,A -85,B 0,C 180,E1 -4036.647,E2 -4036.647} C_VEL
LIN {X 0,Y 539.222,Z 537.441,A -85,B 0,C 180,E1 -4036.888,E2 -4036.888} C_VEL
LIN {X 0,Y 539.054,Z 550.478,A -85,B 0,C 180,E1 -4037.29,E2 -4037.29} C_VEL
LIN {X 0,Y 538.894,Z 561.493,A -85,B 0,C 180,E1 -4037.765,E2 -4037.765} C_VEL
LIN {X 0,Y 538.676,Z 573.661,A -85,B 0,C 180,E1 -4038.451,E2 -4038.451} C_VEL
LIN {X 0,Y 538.381,Z 585.095,A -85,B 0,C 180,E1 -4039.28,E2 -4039.28} C_VEL
LIN {X 0,Y 538.138,Z 595.541,A -85,B 0,C 180,E1 -4040.225,E2 -4040.225} C_VEL
LIN {X 0,Y 537.973,Z 603.993,A -85,B 0,C 180,E1 -4041.17,E2 -4041.17} C_VEL
LIN {X 0,Y 537.816,Z 612.237,A -85,B 0,C 180,E1 -4042.303,E2 -4042.303} C_VEL
LIN {X 0,Y 537.683,Z 618.751,A -85,B 0,C 180,E1 -4043.409,E2 -4043.409} C_VEL
LIN {X 0,Y 537.676,Z 623.367,A -85,B 0,C 180,E1 -4044.374,E2 -4044.374} C_VEL
LIN {X 0,Y 537.557,Z 627.677,A -85,B 0,C 180,E1 -4045.501,E2 -4045.501} C_VEL
LIN {X 0,Y 537.591,Z 629.959,A -85,B 0,C 180,E1 -4046.252,E2 -4046.252} C_VEL
LIN {X 0,Y 537.551,Z 631.808,A -85,B 0,C 180,E1 -4047.002,E2 -4047.002} C_VEL
LIN {X 0,Y 537.451,Z 634.183,A -85,B 0,C 180,E1 -4048.502,E2 -4048.502} C_VEL
LIN {X 0,Y 537.442,Z 635,A -85,B 0,C 180,E1 -4050,E2 -4050} C_VEL
LIN {X 0,Y 537.451,Z 634.184,A -85,B 0,C 180,E1 -4051.499,E2 -4051.499} C_VEL
LIN {X 0,Y 537.551,Z 631.81,A -85,B 0,C 180,E1 -4052.998,E2 -4052.998} C_VEL
LIN {X 0,Y 537.603,Z 628.895,A -85,B 0,C 180,E1 -4054.123,E2 -4054.123} C_VEL
LIN {X 0,Y 537.588,Z 624.948,A -85,B 0,C 180,E1 -4055.251,E2 -4055.251} C_VEL
LIN {X 0,Y 537.65,Z 620.08,A -85,B 0,C 180,E1 -4056.336,E2 -4056.336} C_VEL
LIN {X 0,Y 537.791,Z 613.466,A -85,B 0,C 180,E1 -4057.509,E2 -4057.509} C_VEL
LIN {X 0,Y 537.973,Z 605.476,A -85,B 0,C 180,E1 -4058.641,E2 -4058.641} C_VEL
LIN {X 0,Y 538.119,Z 597.332,A -85,B 0,C 180,E1 -4059.586,E2 -4059.586} C_VEL
LIN {X 0,Y 538.362,Z 587.396,A -85,B 0,C 180,E1 -4060.531,E2 -4060.531} C_VEL
LIN {X 0,Y 538.574,Z 577.588,A -85,B 0,C 180,E1 -4061.288,E2 -4061.288} C_VEL
LIN {X 0,Y 538.763,Z 566.438,A -85,B 0,C 180,E1 -4061.979,E2 -4061.979} C_VEL
LIN {X 0,Y 538.966,Z 554.098,A -85,B 0,C 180,E1 -4062.568,E2 -4062.568} C_VEL
LIN {X 0,Y 539.195,Z 541.079,A -85,B 0,C 180,E1 -4063.018,E2 -4063.018} C_VEL
LIN {X 0,Y 538.954,Z 534.779,A -85,B 0,C 180,E1 -4063.182,E2 -4063.182} C_VEL
LIN {X 0,Y 537.754,Z 527.529,A -85,B 0,C 180,E1 -4063.366,E2 -4063.366} C_VEL
LIN {X 0,Y 537.875,Z 518.759,A -85,B 0,C 180,E1 -4065.926,E2 -4065.926} C_VEL
LIN {X 0,Y 537.966,Z 509.175,A -85,B 0,C 180,E1 -4068.667,E2 -4068.667} C_VEL
LIN {X 0,Y 538.054,Z 499.338,A -85,B 0,C 180,E1 -4071.453,E2 -4071.453} C_VEL
LIN {X 0,Y 538.173,Z 489.717,A -85,B 0,C 180,E1 -4074.29,E2 -4074.29} C_VEL
LIN {X 0,Y 538.337,Z 480.129,A -85,B 0,C 180,E1 -4077.189,E2 -4077.189} C_VEL
LIN {X 0,Y 538.577,Z 469.584,A -85,B 0,C 180,E1 -4080.592,E2 -4080.592} C_VEL
LIN {X 0,Y 538.792,Z 461.688,A -85,B 0,C 180,E1 -4083.403,E2 -4083.403} C_VEL
LIN {X 0,Y 539.05,Z 456.539,A -85,B 0,C 180,E1 -4085.463,E2 -4085.463} C_VEL
LIN {X 0,Y 538.637,Z 452.726,A -85,B 0,C 180,E1 -4087.258,E2 -4087.258} C_VEL
LIN {X 0,Y 538.064,Z 449.465,A -85,B 0,C 180,E1 -4089.188,E2 -4089.188} C_VEL
LIN {X 0,Y 538.035,Z 449.468,A -85,B 0,C 180,E1 -4091.879,E2 -4091.879} C_VEL
LIN {X 0,Y 538.036,Z 449.469,A -85,B 0,C 180,E1 -4095.141,E2 -4095.141} C_VEL
LIN {X 0,Y 538.045,Z 449.466,A -85,B 0,C 180,E1 -4098.228,E2 -4098.228} C_VEL
LIN {X 0,Y 538.019,Z 449.471,A -85,B 0,C 180,E1 -4101.17,E2 -4101.17} C_VEL
LIN {X 0,Y 537.961,Z 449.478,A -85,B 0,C 180,E1 -4103.993,E2 -4103.993} C_VEL
LIN {X 0,Y 537.958,Z 449.634,A -85,B 0,C 180,E1 -4104.913,E2 -4104.913} C_VEL
LIN {X 0,Y 537.922,Z 452.09,A -85,B 0,C 180,E1 -4107.611,E2 -4107.611} C_VEL
LIN {X 0,Y 537.837,Z 454.567,A -85,B 0,C 180,E1 -4110.228,E2 -4110.228} C_VEL
LIN {X 0,Y 537.766,Z 457.041,A -85,B 0,C 180,E1 -4112.78,E2 -4112.78} C_VEL
LIN {X 0,Y 537.718,Z 459.516,A -85,B 0,C 180,E1 -4115.276,E2 -4115.276} C_VEL
LIN {X 0,Y 537.638,Z 462.852,A -85,B 0,C 180,E1 -4118.53,E2 -4118.53} C_VEL
LIN {X 0,Y 537.57,Z 465.316,A -85,B 0,C 180,E1 -4120.923,E2 -4120.923} C_VEL
LIN {X 0,Y 537.548,Z 467.756,A -85,B 0,C 180,E1 -4123.284,E2 -4123.284} C_VEL
LIN {X 0,Y 537.543,Z 470.263,A -85,B 0,C 180,E1 -4125.617,E2 -4125.617} C_VEL
LIN {X 0,Y 537.478,Z 471.674,A -85,B 0,C 180,E1 -4126.748,E2 -4126.748} C_VEL
LIN {X 0,Y 539.189,Z 482.779,A -85,B 0,C 180,E1 -4127.078,E2 -4127.078} C_VEL
LIN {X 0,Y 539.003,Z 495.301,A -85,B 0,C 180,E1 -4127.528,E2 -4127.528} C_VEL
LIN {X 0,Y 538.774,Z 507.531,A -85,B 0,C 180,E1 -4128.126,E2 -4128.126} C_VEL
LIN {X 0,Y 538.558,Z 518.296,A -85,B 0,C 180,E1 -4128.807,E2 -4128.807} C_VEL
LIN {X 0,Y 538.273,Z 529.031,A -85,B 0,C 180,E1 -4129.658,E2 -4129.658} C_VEL
LIN {X 0,Y 538.086,Z 538.693,A -85,B 0,C 180,E1 -4130.604,E2 -4130.604} C_VEL
LIN {X 0,Y 537.923,Z 546.61,A -85,B 0,C 180,E1 -4131.548,E2 -4131.548} C_VEL
LIN {X 0,Y 537.76,Z 554.356,A -85,B 0,C 180,E1 -4132.679,E2 -4132.679} C_VEL
LIN {X 0,Y 537.694,Z 561.463,A -85,B 0,C 180,E1 -4133.998,E2 -4133.998} C_VEL
LIN {X 0,Y 537.54,Z 566.202,A -85,B 0,C 180,E1 -4135.125,E2 -4135.125} C_VEL
LIN {X 0,Y 537.591,Z 569.833,A -85,B 0,C 180,E1 -4136.252,E2 -4136.252} C_VEL
LIN {X 0,Y 537.551,Z 571.709,A -85,B 0,C 180,E1 -4137.002,E2 -4137.002} C_VEL
LIN {X 0,Y 537.489,Z 573.13,A -85,B 0,C 180,E1 -4137.752,E2 -4137.752} C_VEL
LIN {X 0,Y 537.442,Z 574.758,A -85,B 0,C 180,E1 -4139.251,E2 -4139.251} C_VEL
LIN {X 0,Y 537.442,Z 574.996,A -85,B 0,C 180,E1 -4140,E2 -4140} C_VEL
LIN {X 0,Y 537.442,Z 574.814,A -85,B 0,C 180,E1 -4140.749,E2 -4140.749} C_VEL
LIN {X 0,Y 537.489,Z 573.262,A -85,B 0,C 180,E1 -4142.248,E2 -4142.248} C_VEL
LIN {X 0,Y 537.552,Z 571.9,A -85,B 0,C 180,E1 -4142.998,E2 -4142.998} C_VEL
LIN {X 0,Y 537.603,Z 569.022,A -85,B 0,C 180,E1 -4144.123,E2 -4144.123} C_VEL
LIN {X 0,Y 537.587,Z 565.119,A -85,B 0,C 180,E1 -4145.251,E2 -4145.251} C_VEL
LIN {X 0,Y 537.636,Z 560.373,A -85,B 0,C 180,E1 -4146.32,E2 -4146.32} C_VEL
LIN {X 0,Y 537.79,Z 553.755,A -85,B 0,C 180,E1 -4147.509,E2 -4147.509} C_VEL
LIN {X 0,Y 537.952,Z 545.829,A -85,B 0,C 180,E1 -4148.641,E2 -4148.641} C_VEL
LIN {X 0,Y 538.133,Z 535.972,A -85,B 0,C 180,E1 -4149.775,E2 -4149.775} C_VEL
LIN {X 0,Y 538.375,Z 525.644,A -85,B 0,C 180,E1 -4150.721,E2 -4150.721} C_VEL
LIN {X 0,Y 538.622,Z 514.663,A -85,B 0,C 180,E1 -4151.528,E2 -4151.528} C_VEL
LIN {X 0,Y 538.82,Z 504.233,A -85,B 0,C 180,E1 -4152.142,E2 -4152.142} C_VEL
LIN {X 0,Y 539.013,Z 492.908,A -85,B 0,C 180,E1 -4152.663,E2 -4152.663} C_VEL
LIN {X 0,Y 539.021,Z 480.517,A -85,B 0,C 180,E1 -4153.082,E2 -4153.082} C_VEL
LIN {X 0,Y 537.518,Z 471.666,A -85,B 0,C 180,E1 -4153.348,E2 -4153.348} C_VEL
LIN {X 0,Y 537.539,Z 468.531,A -85,B 0,C 180,E1 -4155.936,E2 -4155.936} C_VEL
LIN {X 0,Y 537.542,Z 465.817,A -85,B 0,C 180,E1 -4158.288,E2 -4158.288} C_VEL
LIN {X 0,Y 537.548,Z 463.128,A -85,B 0,C 180,E1 -4160.671,E2 -4160.671} C_VEL
LIN {X 0,Y 537.623,Z 459.714,A -85,B 0,C 180,E1 -4163.784,E2 -4163.784} C_VEL
LIN {X 0,Y 537.668,Z 456.74,A -85,B 0,C 180,E1 -4166.387,E2 -4166.387} C_VEL
LIN {X 0,Y 537.656,Z 453.839,A -85,B 0,C 180,E1 -4168.924,E2 -4168.924} C_VEL
LIN {X 0,Y 537.693,Z 450.628,A -85,B 0,C 180,E1 -4171.832,E2 -4171.832} C_VEL
LIN {X 0,Y 537.768,Z 449.501,A -85,B 0,C 180,E1 -4173.291,E2 -4173.291} C_VEL
LIN {X 0,Y 537.962,Z 449.473,A -85,B 0,C 180,E1 -4176.008,E2 -4176.008} C_VEL
LIN {X 0,Y 537.966,Z 449.472,A -85,B 0,C 180,E1 -4176.269,E2 -4176.269} C_VEL
LIN {X 0,Y 537.329,Z 449.555,A -85,B 0,C 180,E1 -4176.894,E2 -4176.894} C_VEL
LIN {X 0,Y 534.51,Z 449.904,A -85,B 0,C 180,E1 -4177.91,E2 -4177.91} C_VEL
LIN {X 0,Y 532.109,Z 450.203,A -85,B 0,C 180,E1 -4178.727,E2 -4178.727} C_VEL
LIN {X 0,Y 531.072,Z 450.331,A -85,B 0,C 180,E1 -4179.358,E2 -4179.358} C_VEL
LIN {X 0,Y 530.985,Z 450.343,A -85,B 0,C 180,E1 -4179.571,E2 -4179.571} C_VEL
LIN {X 0,Y 530.985,Z 450.343,A -85,B 0,C 180,E1 -4182.457,E2 -4182.457} C_VEL
LIN {X 0,Y 530.982,Z 450.342,A -85,B 0,C 180,E1 -4185.622,E2 -4185.622} C_VEL
LIN {X 0,Y 530.999,Z 450.341,A -85,B 0,C 180,E1 -4188.565,E2 -4188.565} C_VEL
LIN {X 0,Y 530.963,Z 450.345,A -85,B 0,C 180,E1 -4191.53,E2 -4191.53} C_VEL
LIN {X 0,Y 530.961,Z 450.346,A -85,B 0,C 180,E1 -4194.38,E2 -4194.38} C_VEL
LIN {X 0,Y 530.973,Z 450.347,A -85,B 0,C 180,E1 -4197.133,E2 -4197.133} C_VEL
LIN {X 0,Y 530.966,Z 450.345,A -85,B 0,C 180,E1 -4199.803,E2 -4199.803} C_VEL
LIN {X 0,Y 531.016,Z 450.338,A -85,B 0,C 180,E1 -4202.468,E2 -4202.468} C_VEL
LIN {X 0,Y 531.012,Z 450.342,A -85,B 0,C 180,E1 -4204.943,E2 -4204.943} C_VEL
LIN {X 0,Y 530.978,Z 450.345,A -85,B 0,C 180,E1 -4208.247,E2 -4208.247} C_VEL
LIN {X 0,Y 530.999,Z 450.342,A -85,B 0,C 180,E1 -4210.677,E2 -4210.677} C_VEL
LIN {X 0,Y 530.987,Z 450.343,A -85,B 0,C 180,E1 -4213.071,E2 -4213.071} C_VEL
LIN {X 0,Y 531.026,Z 450.338,A -85,B 0,C 180,E1 -4215.436,E2 -4215.436} C_VEL
LIN {X 0,Y 531.044,Z 450.337,A -85,B 0,C 180,E1 -4218.55,E2 -4218.55} C_VEL
LIN {X 0,Y 531.042,Z 450.336,A -85,B 0,C 180,E1 -4221.629,E2 -4221.629} C_VEL
LIN {X 0,Y 531.125,Z 450.326,A -85,B 0,C 180,E1 -4224.685,E2 -4224.685} C_VEL
LIN {X 0,Y 531.145,Z 450.323,A -85,B 0,C 180,E1 -4227.725,E2 -4227.725} C_VEL
LIN {X 0,Y 531.159,Z 450.32,A -85,B 0,C 180,E1 -4230.758,E2 -4230.758} C_VEL
LIN {X 0,Y 531.108,Z 450.331,A -85,B 0,C 180,E1 -4233.034,E2 -4233.034} C_VEL
LIN {X 0,Y 531.072,Z 450.336,A -85,B 0,C 180,E1 -4236.077,E2 -4236.077} C_VEL
LIN {X 0,Y 531.061,Z 450.333,A -85,B 0,C 180,E1 -4238.37,E2 -4238.37} C_VEL
LIN {X 0,Y 531.058,Z 450.333,A -85,B 0,C 180,E1 -4241.672,E2 -4241.672} C_VEL
LIN {X 0,Y 531.037,Z 450.336,A -85,B 0,C 180,E1 -4244.956,E2 -4244.956} C_VEL
LIN {X 0,Y 531.022,Z 450.338,A -85,B 0,C 180,E1 -4247.722,E2 -4247.722} C_VEL
LIN {X 0,Y 531.03,Z 450.341,A -85,B 0,C 180,E1 -4250.127,E2 -4250.127} C_VEL
LIN {X 0,Y 530.951,Z 450.346,A -85,B 0,C 180,E1 -4252.573,E2 -4252.573} C_VEL
LIN {X 0,Y 531.01,Z 450.342,A -85,B 0,C 180,E1 -4255.057,E2 -4255.057} C_VEL
LIN {X 0,Y 531.016,Z 450.34,A -85,B 0,C 180,E1 -4257.595,E2 -4257.595} C_VEL
LIN {X 0,Y 530.979,Z 450.345,A -85,B 0,C 180,E1 -4260.645,E2 -4260.645} C_VEL
LIN {X 0,Y 530.994,Z 450.343,A -85,B 0,C 180,E1 -4263.772,E2 -4263.772} C_VEL
LIN {X 0,Y 530.969,Z 450.344,A -85,B 0,C 180,E1 -4266.557,E2 -4266.557} C_VEL
LIN {X 0,Y 530.981,Z 450.344,A -85,B 0,C 180,E1 -4269.853,E2 -4269.853} C_VEL
LIN {X 0,Y 530.981,Z 450.342,A -85,B 0,C 180,E1 -4272.456,E2 -4272.456} C_VEL
LIN {X 0,Y 530.992,Z 450.342,A -85,B 0,C 180,E1 -4275.62,E2 -4275.62} C_VEL
LIN {X 0,Y 531.001,Z 450.341,A -85,B 0,C 180,E1 -4278.564,E2 -4278.564} C_VEL
LIN {X 0,Y 530.96,Z 450.348,A -85,B 0,C 180,E1 -4281.529,E2 -4281.529} C_VEL
LIN {X 0,Y 530.982,Z 450.346,A -85,B 0,C 180,E1 -4284.382,E2 -4284.382} C_VEL
LIN {X 0,Y 530.972,Z 450.344,A -85,B 0,C 180,E1 -4287.133,E2 -4287.133} C_VEL
LIN {X 0,Y 530.972,Z 450.344,A -85,B 0,C 180,E1 -4289.803,E2 -4289.803} C_VEL
LIN {X 0,Y 531.018,Z 450.34,A -85,B 0,C 180,E1 -4292.466,E2 -4292.466} C_VEL
LIN {X 0,Y 531.008,Z 450.34,A -85,B 0,C 180,E1 -4294.942,E2 -4294.942} C_VEL
LIN {X 0,Y 530.974,Z 450.348,A -85,B 0,C 180,E1 -4298.246,E2 -4298.246} C_VEL
LIN {X 0,Y 530.997,Z 450.34,A -85,B 0,C 180,E1 -4300.677,E2 -4300.677} C_VEL
LIN {X 0,Y 530.988,Z 450.346,A -85,B 0,C 180,E1 -4303.071,E2 -4303.071} C_VEL
LIN {X 0,Y 531.022,Z 450.338,A -85,B 0,C 180,E1 -4305.436,E2 -4305.436} C_VEL
LIN {X 0,Y 531.039,Z 450.334,A -85,B 0,C 180,E1 -4308.55,E2 -4308.55} C_VEL
LIN {X 0,Y 531.058,Z 450.333,A -85,B 0,C 180,E1 -4311.629,E2 -4311.629} C_VEL
LIN {X 0,Y 531.123,Z 450.325,A -85,B 0,C 180,E1 -4314.685,E2 -4314.685} C_VEL
LIN {X 0,Y 531.139,Z 450.323,A -85,B 0,C 180,E1 -4317.725,E2 -4317.725} C_VEL
LIN {X 0,Y 531.155,Z 450.322,A -85,B 0,C 180,E1 -4320.758,E2 -4320.758} C_VEL
LIN {X 0,Y 531.107,Z 450.328,A -85,B 0,C 180,E1 -4323.034,E2 -4323.034} C_VEL
LIN {X 0,Y 531.085,Z 450.331,A -85,B 0,C 180,E1 -4326.077,E2 -4326.077} C_VEL
LIN {X 0,Y 531.029,Z 450.337,A -85,B 0,C 180,E1 -4329.138,E2 -4329.138} C_VEL
LIN {X 0,Y 531.042,Z 450.336,A -85,B 0,C 180,E1 -4332.225,E2 -4332.225} C_VEL
LIN {X 0,Y 530.997,Z 450.342,A -85,B 0,C 180,E1 -4335.35,E2 -4335.35} C_VEL
LIN {X 0,Y 530.992,Z 450.342,A -85,B 0,C 180,E1 -4338.521,E2 -4338.521} C_VEL
LIN {X 0,Y 531.001,Z 450.342,A -85,B 0,C 180,E1 -4340.938,E2 -4340.938} C_VEL
LIN {X 0,Y 530.981,Z 450.342,A -85,B 0,C 180,E1 -4344.224,E2 -4344.224} C_VEL
LIN {X 0,Y 531.006,Z 450.343,A -85,B 0,C 180,E1 -4346.744,E2 -4346.744} C_VEL
LIN {X 0,Y 530.983,Z 450.343,A -85,B 0,C 180,E1 -4349.323,E2 -4349.323} C_VEL
LIN {X 0,Y 530.966,Z 450.344,A -85,B 0,C 180,E1 -4352.1,E2 -4352.1} C_VEL
LIN {X 0,Y 530.986,Z 450.345,A -85,B 0,C 180,E1 -4354.854,E2 -4354.854} C_VEL
LIN {X 0,Y 530.967,Z 450.348,A -85,B 0,C 180,E1 -4357.508,E2 -4357.508} C_VEL
LIN {X 0,Y 530.983,Z 450.344,A -85,B 0,C 180,E1 -4360.433,E2 -4360.433} C_VEL
LIN {X 0,Y 530.972,Z 450.344,A -85,B 0,C 180,E1 -4363.282,E2 -4363.282} C_VEL
LIN {X 0,Y 530.978,Z 450.349,A -85,B 0,C 180,E1 -4365.622,E2 -4365.622} C_VEL
LIN {X 0,Y 530.998,Z 450.346,A -85,B 0,C 180,E1 -4368.565,E2 -4368.565} C_VEL
LIN {X 0,Y 530.984,Z 450.346,A -85,B 0,C 180,E1 -4371.653,E2 -4371.653} C_VEL
LIN {X 0,Y 531.347,Z 452.365,A -85,B 0,C 180,E1 -4372.524,E2 -4372.524} C_VEL
LIN {X 0,Y 532.07,Z 457.507,A -85,B 0,C 180,E1 -4374.466,E2 -4374.466} C_VEL
LIN {X 0,Y 531.904,Z 464.035,A -85,B 0,C 180,E1 -4376.766,E2 -4376.766} C_VEL
LIN {X 0,Y 531.714,Z 471.243,A -85,B 0,C 180,E1 -4379.221,E2 -4379.221} C_VEL
LIN {X 0,Y 531.433,Z 481.003,A -85,B 0,C 180,E1 -4382.428,E2 -4382.428} C_VEL
LIN {X 0,Y 531.235,Z 490.288,A -85,B 0,C 180,E1 -4385.372,E2 -4385.372} C_VEL
LIN {X 0,Y 531.04,Z 500.911,A -85,B 0,C 180,E1 -4388.657,E2 -4388.657} C_VEL
LIN {X 0,Y 530.899,Z 510.448,A -85,B 0,C 180,E1 -4391.476,E2 -4391.476} C_VEL
LIN {X 0,Y 530.798,Z 519.953,A -85,B 0,C 180,E1 -4394.251,E2 -4394.251} C_VEL
LIN {X 0,Y 530.72,Z 527.737,A -85,B 0,C 180,E1 -4396.473,E2 -4396.473} C_VEL
LIN {X 0,Y 532.33,Z 538.356,A -85,B 0,C 180,E1 -4396.739,E2 -4396.739} C_VEL
LIN {X 0,Y 532.118,Z 551.778,A -85,B 0,C 180,E1 -4397.171,E2 -4397.171} C_VEL
LIN {X 0,Y 531.931,Z 563.409,A -85,B 0,C 180,E1 -4397.699,E2 -4397.699} C_VEL
LIN {X 0,Y 531.658,Z 575.809,A -85,B 0,C 180,E1 -4398.442,E2 -4398.442} C_VEL
LIN {X 0,Y 531.384,Z 586.267,A -85,B 0,C 180,E1 -4399.233,E2 -4399.233} C_VEL
LIN {X 0,Y 531.113,Z 595.541,A -85,B 0,C 180,E1 -4400.095,E2 -4400.095} C_VEL
LIN {X 0,Y 530.931,Z 603.993,A -85,B 0,C 180,E1 -4401.052,E2 -4401.052} C_VEL
LIN {X 0,Y 530.758,Z 612.236,A -85,B 0,C 180,E1 -4402.2,E2 -4402.2} C_VEL
LIN {X 0,Y 530.597,Z 619.269,A -85,B 0,C 180,E1 -4403.419,E2 -4403.419} C_VEL
LIN {X 0,Y 530.525,Z 624.95,A -85,B 0,C 180,E1 -4404.679,E2 -4404.679} C_VEL
LIN {X 0,Y 530.522,Z 628.895,A -85,B 0,C 180,E1 -4405.822,E2 -4405.822} C_VEL
LIN {X 0,Y 530.457,Z 631.807,A -85,B 0,C 180,E1 -4406.962,E2 -4406.962} C_VEL
LIN {X 0,Y 530.41,Z 633.194,A -85,B 0,C 180,E1 -4407.722,E2 -4407.722} C_VEL
LIN {X 0,Y 530.344,Z 634.786,A -85,B 0,C 180,E1 -4409.241,E2 -4409.241} C_VEL
LIN {X 0,Y 530.342,Z 635,A -85,B 0,C 180,E1 -4410,E2 -4410} C_VEL
LIN {X 0,Y 530.361,Z 634.184,A -85,B 0,C 180,E1 -4411.519,E2 -4411.519} C_VEL
LIN {X 0,Y 530.41,Z 633.196,A -85,B 0,C 180,E1 -4412.278,E2 -4412.278} C_VEL
LIN {X 0,Y 530.457,Z 631.81,A -85,B 0,C 180,E1 -4413.038,E2 -4413.038} C_VEL
LIN {X 0,Y 530.522,Z 628.895,A -85,B 0,C 180,E1 -4414.178,E2 -4414.178} C_VEL
LIN {X 0,Y 530.525,Z 624.948,A -85,B 0,C 180,E1 -4415.321,E2 -4415.321} C_VEL
LIN {X 0,Y 530.599,Z 619.262,A -85,B 0,C 180,E1 -4416.582,E2 -4416.582} C_VEL
LIN {X 0,Y 530.758,Z 612.234,A -85,B 0,C 180,E1 -4417.801,E2 -4417.801} C_VEL
LIN {X 0,Y 530.931,Z 603.99,A -85,B 0,C 180,E1 -4418.948,E2 -4418.948} C_VEL
LIN {X 0,Y 531.113,Z 595.538,A -85,B 0,C 180,E1 -4419.906,E2 -4419.906} C_VEL
LIN {X 0,Y 531.407,Z 585.089,A -85,B 0,C 180,E1 -4420.863,E2 -4420.863} C_VEL
LIN {X 0,Y 531.675,Z 574.168,A -85,B 0,C 180,E1 -4421.669,E2 -4421.669} C_VEL
LIN {X 0,Y 531.931,Z 563.4,A -85,B 0,C 180,E1 -4422.301,E2 -4422.301} C_VEL
LIN {X 0,Y 532.122,Z 551.758,A -85,B 0,C 180,E1 -4422.83,E2 -4422.83} C_VEL
LIN {X 0,Y 532.302,Z 538.336,A -85,B 0,C 180,E1 -4423.262,E2 -4423.262} C_VEL
LIN {X 0,Y 530.709,Z 527.529,A -85,B 0,C 180,E1 -4423.546,E2 -4423.546} C_VEL
LIN {X 0,Y 530.796,Z 518.456,A -85,B 0,C 180,E1 -4426.144,E2 -4426.144} C_VEL
LIN {X 0,Y 530.89,Z 508.696,A -85,B 0,C 180,E1 -4428.925,E2 -4428.925} C_VEL
LIN {X 0,Y 530.996,Z 498.927,A -85,B 0,C 180,E1 -4431.752,E2 -4431.752} C_VEL
LIN {X 0,Y 531.141,Z 489.322,A -85,B 0,C 180,E1 -4434.633,E2 -4434.633} C_VEL
LIN {X 0,Y 531.316,Z 479.832,A -85,B 0,C 180,E1 -4437.579,E2 -4437.579} C_VEL
LIN {X 0,Y 531.57,Z 470.273,A -85,B 0,C 180,E1 -4440.753,E2 -4440.753} C_VEL
LIN {X 0,Y 531.852,Z 462.239,A -85,B 0,C 180,E1 -4443.711,E2 -4443.711} C_VEL
LIN {X 0,Y 532.105,Z 457.829,A -85,B 0,C 180,E1 -4445.532,E2 -4445.532} C_VEL
LIN {X 0,Y 531.614,Z 453.789,A -85,B 0,C 180,E1 -4447.514,E2 -4447.514} C_VEL
LIN {X 0,Y 531.008,Z 450.344,A -85,B 0,C 180,E1 -4449.647,E2 -4449.647} C_VEL
LIN {X 0,Y 530.982,Z 450.348,A -85,B 0,C 180,E1 -4452.457,E2 -4452.457} C_VEL
LIN {X 0,Y 530.992,Z 450.345,A -85,B 0,C 180,E1 -4455.621,E2 -4455.621} C_VEL
LIN {X 0,Y 531.004,Z 450.345,A -85,B 0,C 180,E1 -4458.565,E2 -4458.565} C_VEL
LIN {X 0,Y 530.963,Z 450.349,A -85,B 0,C 180,E1 -4461.53,E2 -4461.53} C_VEL
LIN {X 0,Y 530.92,Z 450.356,A -85,B 0,C 180,E1 -4464.377,E2 -4464.377} C_VEL
LIN {X 0,Y 530.914,Z 452.045,A -85,B 0,C 180,E1 -4466.509,E2 -4466.509} C_VEL
LIN {X 0,Y 530.832,Z 454.654,A -85,B 0,C 180,E1 -4469.382,E2 -4469.382} C_VEL
LIN {X 0,Y 530.736,Z 457.625,A -85,B 0,C 180,E1 -4472.526,E2 -4472.526} C_VEL
LIN {X 0,Y 530.651,Z 459.965,A -85,B 0,C 180,E1 -4474.925,E2 -4474.925} C_VEL
LIN {X 0,Y 530.573,Z 462.447,A -85,B 0,C 180,E1 -4477.41,E2 -4477.41} C_VEL
LIN {X 0,Y 530.541,Z 465.283,A -85,B 0,C 180,E1 -4480.141,E2 -4480.141} C_VEL
LIN {X 0,Y 530.501,Z 468.236,A -85,B 0,C 180,E1 -4483.055,E2 -4483.055} C_VEL
LIN {X 0,Y 530.487,Z 470.731,A -85,B 0,C 180,E1 -4485.421,E2 -4485.421} C_VEL
LIN {X 0,Y 530.43,Z 471.979,A -85,B 0,C 180,E1 -4486.569,E2 -4486.569} C_VEL
LIN {X 0,Y 532.262,Z 483.592,A -85,B 0,C 180,E1 -4486.931,E2 -4486.931} C_VEL
LIN {X 0,Y 532.044,Z 496.462,A -85,B 0,C 180,E1 -4487.411,E2 -4487.411} C_VEL
LIN {X 0,Y 531.803,Z 508.684,A -85,B 0,C 180,E1 -4488.035,E2 -4488.035} C_VEL
LIN {X 0,Y 531.556,Z 519.593,A -85,B 0,C 180,E1 -4488.754,E2 -4488.754} C_VEL
LIN {X 0,Y 531.258,Z 530.105,A -85,B 0,C 180,E1 -4489.616,E2 -4489.616} C_VEL
LIN {X 0,Y 531.07,Z 538.698,A -85,B 0,C 180,E1 -4490.478,E2 -4490.478} C_VEL
LIN {X 0,Y 530.891,Z 546.614,A -85,B 0,C 180,E1 -4491.435,E2 -4491.435} C_VEL
LIN {X 0,Y 530.691,Z 554.36,A -85,B 0,C 180,E1 -4492.581,E2 -4492.581} C_VEL
LIN {X 0,Y 530.606,Z 561.466,A -85,B 0,C 180,E1 -4493.918,E2 -4493.918} C_VEL
LIN {X 0,Y 530.459,Z 566.204,A -85,B 0,C 180,E1 -4495.06,E2 -4495.06} C_VEL
LIN {X 0,Y 530.516,Z 569.835,A -85,B 0,C 180,E1 -4496.202,E2 -4496.202} C_VEL
LIN {X 0,Y 530.457,Z 571.711,A -85,B 0,C 180,E1 -4496.962,E2 -4496.962} C_VEL
LIN {X 0,Y 530.41,Z 573.13,A -85,B 0,C 180,E1 -4497.722,E2 -4497.722} C_VEL
LIN {X 0,Y 530.344,Z 574.758,A -85,B 0,C 180,E1 -4499.241,E2 -4499.241} C_VEL
LIN {X 0,Y 530.343,Z 574.997,A -85,B 0,C 180,E1 -4500,E2 -4500} C_VEL
LIN {X 0,Y 530.344,Z 574.814,A -85,B 0,C 180,E1 -4500.759,E2 -4500.759} C_VEL
LIN {X 0,Y 530.41,Z 573.26,A -85,B 0,C 180,E1 -4502.278,E2 -4502.278} C_VEL
LIN {X 0,Y 530.458,Z 571.898,A -85,B 0,C 180,E1 -4503.038,E2 -4503.038} C_VEL
LIN {X 0,Y 530.523,Z 569.02,A -85,B 0,C 180,E1 -4504.178,E2 -4504.178} C_VEL
LIN {X 0,Y 530.523,Z 565.117,A -85,B 0,C 180,E1 -4505.321,E2 -4505.321} C_VEL
LIN {X 0,Y 530.605,Z 559.088,A -85,B 0,C 180,E1 -4506.66,E2 -4506.66} C_VEL
LIN {X 0,Y 530.758,Z 552.523,A -85,B 0,C 180,E1 -4507.801,E2 -4507.801} C_VEL
LIN {X 0,Y 530.903,Z 544.338,A -85,B 0,C 180,E1 -4508.949,E2 -4508.949} C_VEL
LIN {X 0,Y 531.107,Z 535.966,A -85,B 0,C 180,E1 -4509.906,E2 -4509.906} C_VEL
LIN {X 0,Y 531.399,Z 525.635,A -85,B 0,C 180,E1 -4510.863,E2 -4510.863} C_VEL
LIN {X 0,Y 531.652,Z 513.9,A -85,B 0,C 180,E1 -4511.732,E2 -4511.732} C_VEL
LIN {X 0,Y 531.904,Z 502.41,A -85,B 0,C 180,E1 -4512.399,E2 -4512.399} C_VEL
LIN {X 0,Y 532.134,Z 490.389,A -85,B 0,C 180,E1 -4512.927,E2 -4512.927} C_VEL
LIN {X 0,Y 532.087,Z 481.415,A -85,B 0,C 180,E1 -4513.231,E2 -4513.231} C_VEL
LIN {X 0,Y 530.419,Z 471.776,A -85,B 0,C 180,E1 -4513.53,E2 -4513.53} C_VEL
LIN {X 0,Y 530.446,Z 468.724,A -85,B 0,C 180,E1 -4516.155,E2 -4516.155} C_VEL
LIN {X 0,Y 530.471,Z 465.114,A -85,B 0,C 180,E1 -4519.343,E2 -4519.343} C_VEL
LIN {X 0,Y 530.496,Z 462.221,A -85,B 0,C 180,E1 -4521.973,E2 -4521.973} C_VEL
LIN {X 0,Y 530.529,Z 458.789,A -85,B 0,C 180,E1 -4525.082,E2 -4525.082} C_VEL
LIN {X 0,Y 530.58,Z 455.927,A -85,B 0,C 180,E1 -4527.62,E2 -4527.62} C_VEL
LIN {X 0,Y 530.613,Z 452.649,A -85,B 0,C 180,E1 -4530.579,E2 -4530.579} C_VEL
LIN {X 0,Y 530.649,Z 450.389,A -85,B 0,C 180,E1 -4532.889,E2 -4532.889} C_VEL
LIN {X 0,Y 530.89,Z 450.358,A -85,B 0,C 180,E1 -4534.838,E2 -4534.838} C_VEL
LIN {X 0,Y 530.969,Z 450.344,A -85,B 0,C 180,E1 -4537.508,E2 -4537.508} C_VEL
LIN {X 0,Y 530.985,Z 450.343,A -85,B 0,C 180,E1 -4539.571,E2 -4539.571} C_VEL
LIN {X 0,Y 530.31,Z 450.431,A -85,B 0,C 180,E1 -4540.204,E2 -4540.204} C_VEL
LIN {X 0,Y 527.449,Z 450.785,A -85,B 0,C 180,E1 -4541.232,E2 -4541.232} C_VEL
LIN {X 0,Y 525.038,Z 451.084,A -85,B 0,C 180,E1 -4542.059,E2 -4542.059} C_VEL
LIN {X 0,Y 524.006,Z 451.214,A -85,B 0,C 180,E1 -4542.698,E2 -4542.698} C_VEL
LIN {X 0,Y 523.924,Z 451.223,A -85,B 0,C 180,E1 -4542.914,E2 -4542.914} C_VEL
LIN {X 0,Y 523.937,Z 451.221,A -85,B 0,C 180,E1 -4545.771,E2 -4545.771} C_VEL
LIN {X 0,Y 523.944,Z 451.221,A -85,B 0,C 180,E1 -4548.908,E2 -4548.908} C_VEL
LIN {X 0,Y 523.921,Z 451.223,A -85,B 0,C 180,E1 -4551.898,E2 -4551.898} C_VEL
LIN {X 0,Y 523.931,Z 451.221,A -85,B 0,C 180,E1 -4554.911,E2 -4554.911} C_VEL
LIN {X 0,Y 523.941,Z 451.22,A -85,B 0,C 180,E1 -4557.68,E2 -4557.68} C_VEL
LIN {X 0,Y 523.958,Z 451.218,A -85,B 0,C 180,E1 -4560.677,E2 -4560.677} C_VEL
LIN {X 0,Y 523.979,Z 451.217,A -85,B 0,C 180,E1 -4563.729,E2 -4563.729} C_VEL
LIN {X 0,Y 523.932,Z 451.224,A -85,B 0,C 180,E1 -4566.27,E2 -4566.27} C_VEL
LIN {X 0,Y 523.952,Z 451.218,A -85,B 0,C 180,E1 -4568.767,E2 -4568.767} C_VEL
LIN {X 0,Y 523.956,Z 451.221,A -85,B 0,C 180,E1 -4571.221,E2 -4571.221} C_VEL
LIN {X 0,Y 523.938,Z 451.22,A -85,B 0,C 180,E1 -4573.639,E2 -4573.639} C_VEL
LIN {X 0,Y 523.946,Z 451.222,A -85,B 0,C 180,E1 -4576.028,E2 -4576.028} C_VEL
LIN {X 0,Y 524.019,Z 451.211,A -85,B 0,C 180,E1 -4578.394,E2 -4578.394} C_VEL
LIN {X 0,Y 523.994,Z 451.213,A -85,B 0,C 180,E1 -4581.516,E2 -4581.516} C_VEL
LIN {X 0,Y 524.051,Z 451.209,A -85,B 0,C 180,E1 -4583.841,E2 -4583.841} C_VEL
LIN {X 0,Y 524.075,Z 451.206,A -85,B 0,C 180,E1 -4586.925,E2 -4586.925} C_VEL
LIN {X 0,Y 524.121,Z 451.201,A -85,B 0,C 180,E1 -4590,E2 -4590} C_VEL
LIN {X 0,Y 524.075,Z 451.206,A -85,B 0,C 180,E1 -4593.075,E2 -4593.075} C_VEL
LIN {X 0,Y 524.031,Z 451.212,A -85,B 0,C 180,E1 -4596.159,E2 -4596.159} C_VEL
LIN {X 0,Y 524.01,Z 451.211,A -85,B 0,C 180,E1 -4598.484,E2 -4598.484} C_VEL
LIN {X 0,Y 524.009,Z 451.212,A -85,B 0,C 180,E1 -4601.739,E2 -4601.739} C_VEL
LIN {X 0,Y 523.999,Z 451.214,A -85,B 0,C 180,E1 -4605.052,E2 -4605.052} C_VEL
LIN {X 0,Y 523.969,Z 451.217,A -85,B 0,C 180,E1 -4607.969,E2 -4607.969} C_VEL
LIN {X 0,Y 523.977,Z 451.216,A -85,B 0,C 180,E1 -4610.41,E2 -4610.41} C_VEL
LIN {X 0,Y 523.917,Z 451.225,A -85,B 0,C 180,E1 -4612.893,E2 -4612.893} C_VEL
LIN {X 0,Y 523.958,Z 451.218,A -85,B 0,C 180,E1 -4615.418,E2 -4615.418} C_VEL
LIN {X 0,Y 523.971,Z 451.219,A -85,B 0,C 180,E1 -4617.999,E2 -4617.999} C_VEL
LIN {X 0,Y 523.949,Z 451.222,A -85,B 0,C 180,E1 -4620.854,E2 -4620.854} C_VEL
LIN {X 0,Y 523.965,Z 451.218,A -85,B 0,C 180,E1 -4623.734,E2 -4623.734} C_VEL
LIN {X 0,Y 523.923,Z 451.222,A -85,B 0,C 180,E1 -4626.403,E2 -4626.403} C_VEL
LIN {X 0,Y 523.924,Z 451.225,A -85,B 0,C 180,E1 -4629.084,E2 -4629.084} C_VEL
LIN {X 0,Y 523.955,Z 451.22,A -85,B 0,C 180,E1 -4632.119,E2 -4632.119} C_VEL
LIN {X 0,Y 523.96,Z 451.22,A -85,B 0,C 180,E1 -4635.308,E2 -4635.308} C_VEL
LIN {X 0,Y 523.962,Z 451.217,A -85,B 0,C 180,E1 -4638.689,E2 -4638.689} C_VEL
LIN {X 0,Y 523.919,Z 451.225,A -85,B 0,C 180,E1 -4641.08,E2 -4641.08} C_VEL
LIN {X 0,Y 523.929,Z 451.222,A -85,B 0,C 180,E1 -4643.827,E2 -4643.827} C_VEL
LIN {X 0,Y 523.945,Z 451.218,A -85,B 0,C 180,E1 -4646.635,E2 -4646.635} C_VEL
LIN {X 0,Y 523.959,Z 451.22,A -85,B 0,C 180,E1 -4649.355,E2 -4649.355} C_VEL
LIN {X 0,Y 523.982,Z 451.218,A -85,B 0,C 180,E1 -4652.281,E2 -4652.281} C_VEL
LIN {X 0,Y 523.955,Z 451.217,A -85,B 0,C 180,E1 -4654.581,E2 -4654.581} C_VEL
LIN {X 0,Y 523.914,Z 451.226,A -85,B 0,C 180,E1 -4657.106,E2 -4657.106} C_VEL
LIN {X 0,Y 523.981,Z 451.219,A -85,B 0,C 180,E1 -4659.866,E2 -4659.866} C_VEL
LIN {X 0,Y 523.969,Z 451.218,A -85,B 0,C 180,E1 -4662.837,E2 -4662.837} C_VEL
LIN {X 0,Y 523.979,Z 451.216,A -85,B 0,C 180,E1 -4665.235,E2 -4665.235} C_VEL
LIN {X 0,Y 524.014,Z 451.209,A -85,B 0,C 180,E1 -4668.394,E2 -4668.394} C_VEL
LIN {X 0,Y 524.007,Z 451.212,A -85,B 0,C 180,E1 -4671.516,E2 -4671.516} C_VEL
LIN {X 0,Y 524.084,Z 451.202,A -85,B 0,C 180,E1 -4674.613,E2 -4674.613} C_VEL
LIN {X 0,Y 524.111,Z 451.199,A -85,B 0,C 180,E1 -4677.694,E2 -4677.694} C_VEL
LIN {X 0,Y 524.125,Z 451.197,A -85,B 0,C 180,E1 -4680.768,E2 -4680.768} C_VEL
LIN {X 0,Y 524.073,Z 451.204,A -85,B 0,C 180,E1 -4683.075,E2 -4683.075} C_VEL
LIN {X 0,Y 524.047,Z 451.209,A -85,B 0,C 180,E1 -4686.159,E2 -4686.159} C_VEL
LIN {X 0,Y 523.997,Z 451.214,A -85,B 0,C 180,E1 -4689.262,E2 -4689.262} C_VEL
LIN {X 0,Y 524.004,Z 451.212,A -85,B 0,C 180,E1 -4691.739,E2 -4691.739} C_VEL
LIN {X 0,Y 523.994,Z 451.213,A -85,B 0,C 180,E1 -4695.052,E2 -4695.052} C_VEL
LIN {X 0,Y 523.965,Z 451.216,A -85,B 0,C 180,E1 -4697.969,E2 -4697.969} C_VEL
LIN {X 0,Y 523.973,Z 451.219,A -85,B 0,C 180,E1 -4700.41,E2 -4700.41} C_VEL
LIN {X 0,Y 523.916,Z 451.223,A -85,B 0,C 180,E1 -4702.893,E2 -4702.893} C_VEL
LIN {X 0,Y 523.954,Z 451.221,A -85,B 0,C 180,E1 -4705.419,E2 -4705.419} C_VEL
LIN {X 0,Y 523.97,Z 451.218,A -85,B 0,C 180,E1 -4707.999,E2 -4707.999} C_VEL
LIN {X 0,Y 523.945,Z 451.219,A -85,B 0,C 180,E1 -4710.855,E2 -4710.855} C_VEL
LIN {X 0,Y 523.961,Z 451.217,A -85,B 0,C 180,E1 -4713.735,E2 -4713.735} C_VEL
LIN {X 0,Y 523.923,Z 451.224,A -85,B 0,C 180,E1 -4716.404,E2 -4716.404} C_VEL
LIN {X 0,Y 523.921,Z 451.225,A -85,B 0,C 180,E1 -4719.085,E2 -4719.085} C_VEL
LIN {X 0,Y 523.958,Z 451.221,A -85,B 0,C 180,E1 -4722.118,E2 -4722.118} C_VEL
LIN {X 0,Y 523.945,Z 451.225,A -85,B 0,C 180,E1 -4725.31,E2 -4725.31} C_VEL
LIN {X 0,Y 523.96,Z 451.222,A -85,B 0,C 180,E1 -4728.689,E2 -4728.689} C_VEL
LIN {X 0,Y 523.948,Z 451.352,A -85,B 0,C 180,E1 -4731.534,E2 -4731.534} C_VEL
LIN {X 0,Y 525.015,Z 457.458,A -85,B 0,C 180,E1 -4733.914,E2 -4733.914} C_VEL
LIN {X 0,Y 525.061,Z 462.615,A -85,B 0,C 180,E1 -4735.794,E2 -4735.794} C_VEL
LIN {X 0,Y 524.789,Z 470.408,A -85,B 0,C 180,E1 -4738.514,E2 -4738.514} C_VEL
LIN {X 0,Y 524.505,Z 478.25,A -85,B 0,C 180,E1 -4741.16,E2 -4741.16} C_VEL
LIN {X 0,Y 524.283,Z 486.68,A -85,B 0,C 180,E1 -4743.914,E2 -4743.914} C_VEL
LIN {X 0,Y 524.077,Z 495.447,A -85,B 0,C 180,E1 -4746.697,E2 -4746.697} C_VEL
LIN {X 0,Y 523.922,Z 504.759,A -85,B 0,C 180,E1 -4749.588,E2 -4749.588} C_VEL
LIN {X 0,Y 523.795,Z 513.845,A -85,B 0,C 180,E1 -4752.296,E2 -4752.296} C_VEL
LIN {X 0,Y 523.714,Z 523.783,A -85,B 0,C 180,E1 -4755.228,E2 -4755.228} C_VEL
LIN {X 0,Y 523.658,Z 527.614,A -85,B 0,C 180,E1 -4756.293,E2 -4756.293} C_VEL
LIN {X 0,Y 525.399,Z 538.956,A -85,B 0,C 180,E1 -4756.585,E2 -4756.585} C_VEL
LIN {X 0,Y 525.186,Z 551.524,A -85,B 0,C 180,E1 -4756.998,E2 -4756.998} C_VEL
LIN {X 0,Y 524.984,Z 563.237,A -85,B 0,C 180,E1 -4757.534,E2 -4757.534} C_VEL
LIN {X 0,Y 524.706,Z 574.334,A -85,B 0,C 180,E1 -4758.192,E2 -4758.192} C_VEL
LIN {X 0,Y 524.431,Z 585.082,A -85,B 0,C 180,E1 -4758.991,E2 -4758.991} C_VEL
LIN {X 0,Y 524.094,Z 595.541,A -85,B 0,C 180,E1 -4759.961,E2 -4759.961} C_VEL
LIN {X 0,Y 523.896,Z 603.993,A -85,B 0,C 180,E1 -4760.931,E2 -4760.931} C_VEL
LIN {X 0,Y 523.688,Z 612.236,A -85,B 0,C 180,E1 -4762.094,E2 -4762.094} C_VEL
LIN {X 0,Y 523.574,Z 617.869,A -85,B 0,C 180,E1 -4763.061,E2 -4763.061} C_VEL
LIN {X 0,Y 523.544,Z 623.367,A -85,B 0,C 180,E1 -4764.222,E2 -4764.222} C_VEL
LIN {X 0,Y 523.361,Z 627.677,A -85,B 0,C 180,E1 -4765.379,E2 -4765.379} C_VEL
LIN {X 0,Y 523.443,Z 629.958,A -85,B 0,C 180,E1 -4766.151,E2 -4766.151} C_VEL
LIN {X 0,Y 523.367,Z 631.807,A -85,B 0,C 180,E1 -4766.921,E2 -4766.921} C_VEL
LIN {X 0,Y 523.334,Z 633.193,A -85,B 0,C 180,E1 -4767.691,E2 -4767.691} C_VEL
LIN {X 0,Y 523.25,Z 634.786,A -85,B 0,C 180,E1 -4769.231,E2 -4769.231} C_VEL
LIN {X 0,Y 523.246,Z 635,A -85,B 0,C 180,E1 -4770,E2 -4770} C_VEL
LIN {X 0,Y 523.274,Z 634.183,A -85,B 0,C 180,E1 -4771.539,E2 -4771.539} C_VEL
LIN {X 0,Y 523.334,Z 633.196,A -85,B 0,C 180,E1 -4772.309,E2 -4772.309} C_VEL
LIN {X 0,Y 523.367,Z 631.81,A -85,B 0,C 180,E1 -4773.079,E2 -4773.079} C_VEL
LIN {X 0,Y 523.441,Z 628.895,A -85,B 0,C 180,E1 -4774.235,E2 -4774.235} C_VEL
LIN {X 0,Y 523.464,Z 624.947,A -85,B 0,C 180,E1 -4775.393,E2 -4775.393} C_VEL
LIN {X 0,Y 523.523,Z 619.726,A -85,B 0,C 180,E1 -4776.581,E2 -4776.581} C_VEL
LIN {X 0,Y 523.665,Z 613.465,A -85,B 0,C 180,E1 -4777.713,E2 -4777.713} C_VEL
LIN {X 0,Y 523.857,Z 605.475,A -85,B 0,C 180,E1 -4778.875,E2 -4778.875} C_VEL
LIN {X 0,Y 524.085,Z 597.331,A -85,B 0,C 180,E1 -4779.845,E2 -4779.845} C_VEL
LIN {X 0,Y 524.363,Z 587.391,A -85,B 0,C 180,E1 -4780.815,E2 -4780.815} C_VEL
LIN {X 0,Y 524.612,Z 577.514,A -85,B 0,C 180,E1 -4781.593,E2 -4781.593} C_VEL
LIN {X 0,Y 524.886,Z 566.017,A -85,B 0,C 180,E1 -4782.312,E2 -4782.312} C_VEL
LIN {X 0,Y 525.123,Z 553.771,A -85,B 0,C 180,E1 -4782.905,E2 -4782.905} C_VEL
LIN {X 0,Y 525.36,Z 540.622,A -85,B 0,C 180,E1 -4783.367,E2 -4783.367} C_VEL
LIN {X 0,Y 524.994,Z 535.996,A -85,B 0,C 180,E1 -4783.499,E2 -4783.499} C_VEL
LIN {X 0,Y 523.642,Z 527.15,A -85,B 0,C 180,E1 -4783.733,E2 -4783.733} C_VEL
LIN {X 0,Y 523.699,Z 517.981,A -85,B 0,C 180,E1 -4786.369,E2 -4786.369} C_VEL
LIN {X 0,Y 523.809,Z 508.215,A -85,B 0,C 180,E1 -4789.191,E2 -4789.191} C_VEL
LIN {X 0,Y 523.929,Z 499.908,A -85,B 0,C 180,E1 -4791.647,E2 -4791.647} C_VEL
LIN {X 0,Y 524.072,Z 490.306,A -85,B 0,C 180,E1 -4794.565,E2 -4794.565} C_VEL
LIN {X 0,Y 524.266,Z 481.195,A -85,B 0,C 180,E1 -4797.446,E2 -4797.446} C_VEL
LIN {X 0,Y 524.536,Z 471.858,A -85,B 0,C 180,E1 -4800.607,E2 -4800.607} C_VEL
LIN {X 0,Y 524.813,Z 464.621,A -85,B 0,C 180,E1 -4803.302,E2 -4803.302} C_VEL
LIN {X 0,Y 525.136,Z 459.841,A -85,B 0,C 180,E1 -4805.276,E2 -4805.276} C_VEL
LIN {X 0,Y 524.825,Z 456.188,A -85,B 0,C 180,E1 -4807.057,E2 -4807.057} C_VEL
LIN {X 0,Y 524.241,Z 452.776,A -85,B 0,C 180,E1 -4809.057,E2 -4809.057} C_VEL
LIN {X 0,Y 523.956,Z 451.222,A -85,B 0,C 180,E1 -4810.33,E2 -4810.33} C_VEL
LIN {X 0,Y 523.925,Z 451.226,A -85,B 0,C 180,E1 -4813.167,E2 -4813.167} C_VEL
LIN {X 0,Y 523.945,Z 451.223,A -85,B 0,C 180,E1 -4815.772,E2 -4815.772} C_VEL
LIN {X 0,Y 523.948,Z 451.223,A -85,B 0,C 180,E1 -4818.908,E2 -4818.908} C_VEL
LIN {X 0,Y 523.92,Z 451.227,A -85,B 0,C 180,E1 -4821.898,E2 -4821.898} C_VEL
LIN {X 0,Y 523.874,Z 451.233,A -85,B 0,C 180,E1 -4823.823,E2 -4823.823} C_VEL
LIN {X 0,Y 523.902,Z 451.733,A -85,B 0,C 180,E1 -4824.915,E2 -4824.915} C_VEL
LIN {X 0,Y 523.851,Z 454.069,A -85,B 0,C 180,E1 -4827.695,E2 -4827.695} C_VEL
LIN {X 0,Y 523.752,Z 456.345,A -85,B 0,C 180,E1 -4830.232,E2 -4830.232} C_VEL
LIN {X 0,Y 523.659,Z 458.772,A -85,B 0,C 180,E1 -4832.851,E2 -4832.851} C_VEL
LIN {X 0,Y 523.604,Z 461.709,A -85,B 0,C 180,E1 -4835.885,E2 -4835.885} C_VEL
LIN {X 0,Y 523.502,Z 464.558,A -85,B 0,C 180,E1 -4838.748,E2 -4838.748} C_VEL
LIN {X 0,Y 523.445,Z 467.092,A -85,B 0,C 180,E1 -4841.202,E2 -4841.202} C_VEL
LIN {X 0,Y 523.421,Z 469.54,A -85,B 0,C 180,E1 -4843.622,E2 -4843.622} C_VEL
LIN {X 0,Y 523.39,Z 472.501,A -85,B 0,C 180,E1 -4846.409,E2 -4846.409} C_VEL
LIN {X 0,Y 525.351,Z 483.781,A -85,B 0,C 180,E1 -4846.756,E2 -4846.756} C_VEL
LIN {X 0,Y 525.115,Z 496.677,A -85,B 0,C 180,E1 -4847.242,E2 -4847.242} C_VEL
LIN {X 0,Y 524.89,Z 507.744,A -85,B 0,C 180,E1 -4847.805,E2 -4847.805} C_VEL
LIN {X 0,Y 524.622,Z 518.543,A -85,B 0,C 180,E1 -4848.506,E2 -4848.506} C_VEL
LIN {X 0,Y 524.298,Z 529.248,A -85,B 0,C 180,E1 -4849.379,E2 -4849.379} C_VEL
LIN {X 0,Y 524.059,Z 538.866,A -85,B 0,C 180,E1 -4850.35,E2 -4850.35} C_VEL
LIN {X 0,Y 523.859,Z 546.736,A -85,B 0,C 180,E1 -4851.319,E2 -4851.319} C_VEL
LIN {X 0,Y 523.638,Z 554.426,A -85,B 0,C 180,E1 -4852.481,E2 -4852.481} C_VEL
LIN {X 0,Y 523.519,Z 561.469,A -85,B 0,C 180,E1 -4853.835,E2 -4853.835} C_VEL
LIN {X 0,Y 523.384,Z 566.206,A -85,B 0,C 180,E1 -4854.993,E2 -4854.993} C_VEL
LIN {X 0,Y 523.444,Z 569.836,A -85,B 0,C 180,E1 -4856.151,E2 -4856.151} C_VEL
LIN {X 0,Y 523.368,Z 571.713,A -85,B 0,C 180,E1 -4856.921,E2 -4856.921} C_VEL
LIN {X 0,Y 523.334,Z 573.13,A -85,B 0,C 180,E1 -4857.691,E2 -4857.691} C_VEL
LIN {X 0,Y 523.25,Z 574.758,A -85,B 0,C 180,E1 -4859.231,E2 -4859.231} C_VEL
LIN {X 0,Y 523.247,Z 574.997,A -85,B 0,C 180,E1 -4860,E2 -4860} C_VEL
LIN {X 0,Y 523.25,Z 574.813,A -85,B 0,C 180,E1 -4860.77,E2 -4860.77} C_VEL
LIN {X 0,Y 523.334,Z 573.258,A -85,B 0,C 180,E1 -4862.309,E2 -4862.309} C_VEL
LIN {X 0,Y 523.368,Z 571.896,A -85,B 0,C 180,E1 -4863.079,E2 -4863.079} C_VEL
LIN {X 0,Y 523.442,Z 569.018,A -85,B 0,C 180,E1 -4864.235,E2 -4864.235} C_VEL
LIN {X 0,Y 523.462,Z 565.115,A -85,B 0,C 180,E1 -4865.393,E2 -4865.393} C_VEL
LIN {X 0,Y 523.53,Z 559.479,A -85,B 0,C 180,E1 -4866.673,E2 -4866.673} C_VEL
LIN {X 0,Y 523.691,Z 552.578,A -85,B 0,C 180,E1 -4867.907,E2 -4867.907} C_VEL
LIN {X 0,Y 523.869,Z 544.443,A -85,B 0,C 180,E1 -4869.07,E2 -4869.07} C_VEL
LIN {X 0,Y 524.097,Z 536.101,A -85,B 0,C 180,E1 -4870.04,E2 -4870.04} C_VEL
LIN {X 0,Y 524.42,Z 525.787,A -85,B 0,C 180,E1 -4871.01,E2 -4871.01} C_VEL
LIN {X 0,Y 524.68,Z 514.639,A -85,B 0,C 180,E1 -4871.851,E2 -4871.851} C_VEL
LIN {X 0,Y 524.925,Z 504.379,A -85,B 0,C 180,E1 -4872.468,E2 -4872.468} C_VEL
LIN {X 0,Y 525.171,Z 493.04,A -85,B 0,C 180,E1 -4873.003,E2 -4873.003} C_VEL
LIN {X 0,Y 525.171,Z 482.319,A -85,B 0,C 180,E1 -4873.384,E2 -4873.384} C_VEL
LIN {X 0,Y 523.367,Z 472.121,A -85,B 0,C 180,E1 -4873.691,E2 -4873.691} C_VEL
LIN {X 0,Y 523.359,Z 469.005,A -85,B 0,C 180,E1 -4876.38,E2 -4876.38} C_VEL
LIN {X 0,Y 523.406,Z 465.387,A -85,B 0,C 180,E1 -4879.615,E2 -4879.615} C_VEL
LIN {X 0,Y 523.409,Z 461.781,A -85,B 0,C 180,E1 -4882.917,E2 -4882.917} C_VEL
LIN {X 0,Y 523.53,Z 458.467,A -85,B 0,C 180,E1 -4885.917,E2 -4885.917} C_VEL
LIN {X 0,Y 523.521,Z 455.122,A -85,B 0,C 180,E1 -4888.9,E2 -4888.9} C_VEL
LIN {X 0,Y 523.558,Z 452.214,A -85,B 0,C 180,E1 -4891.569,E2 -4891.569} C_VEL
LIN {X 0,Y 523.557,Z 451.272,A -85,B 0,C 180,E1 -4892.476,E2 -4892.476} C_VEL
LIN {X 0,Y 523.858,Z 451.233,A -85,B 0,C 180,E1 -4895.232,E2 -4895.232} C_VEL
LIN {X 0,Y 523.919,Z 451.224,A -85,B 0,C 180,E1 -4898.102,E2 -4898.102} C_VEL
LIN {X 0,Y 523.947,Z 451.22,A -85,B 0,C 180,E1 -4901.092,E2 -4901.092} C_VEL
LIN {X 0,Y 523.924,Z 451.223,A -85,B 0,C 180,E1 -4902.914,E2 -4902.914} C_VEL
LIN {X 0,Y 523.265,Z 451.309,A -85,B 0,C 180,E1 -4903.556,E2 -4903.556} C_VEL
LIN {X 0,Y 520.425,Z 451.667,A -85,B 0,C 180,E1 -4904.598,E2 -4904.598} C_VEL
LIN {X 0,Y 518.012,Z 451.966,A -85,B 0,C 180,E1 -4905.437,E2 -4905.437} C_VEL
LIN {X 0,Y 516.965,Z 452.092,A -85,B 0,C 180,E1 -4906.085,E2 -4906.085} C_VEL
LIN {X 0,Y 516.873,Z 452.102,A -85,B 0,C 180,E1 -4906.304,E2 -4906.304} C_VEL
LIN {X 0,Y 516.888,Z 452.101,A -85,B 0,C 180,E1 -4909.258,E2 -4909.258} C_VEL
LIN {X 0,Y 516.869,Z 452.105,A -85,B 0,C 180,E1 -4912.274,E2 -4912.274} C_VEL
LIN {X 0,Y 516.89,Z 452.1,A -85,B 0,C 180,E1 -4915.175,E2 -4915.175} C_VEL
LIN {X 0,Y 516.879,Z 452.1,A -85,B 0,C 180,E1 -4917.975,E2 -4917.975} C_VEL
LIN {X 0,Y 516.926,Z 452.093,A -85,B 0,C 180,E1 -4920.695,E2 -4920.695} C_VEL
LIN {X 0,Y 516.948,Z 452.092,A -85,B 0,C 180,E1 -4923.804,E2 -4923.804} C_VEL
LIN {X 0,Y 516.872,Z 452.101,A -85,B 0,C 180,E1 -4926.776,E2 -4926.776} C_VEL
LIN {X 0,Y 516.946,Z 452.095,A -85,B 0,C 180,E1 -4929.732,E2 -4929.732} C_VEL
LIN {X 0,Y 516.926,Z 452.098,A -85,B 0,C 180,E1 -4932.596,E2 -4932.596} C_VEL
LIN {X 0,Y 516.949,Z 452.089,A -85,B 0,C 180,E1 -4935.03,E2 -4935.03} C_VEL
LIN {X 0,Y 516.972,Z 452.088,A -85,B 0,C 180,E1 -4938.234,E2 -4938.234} C_VEL
